KUKA KRL program: MyProgram_127().src

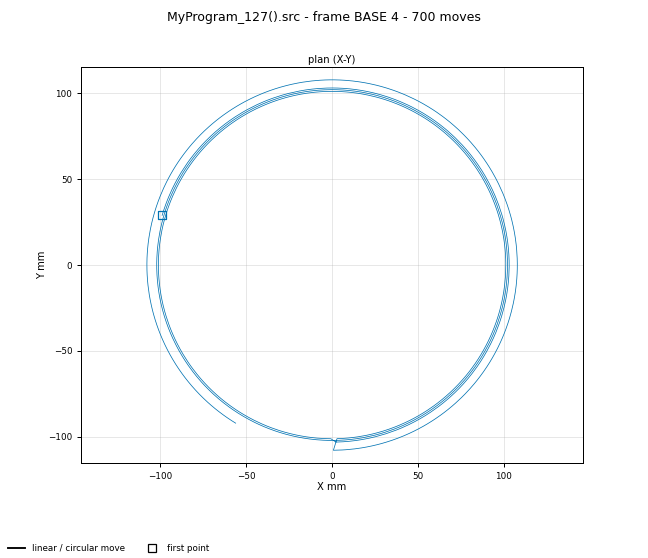
[picture p0: tool path of MyProgram_127().src in frame BASE 4, 700 of 700 moves have a stored position in this frame; points joined in program order, loops and branches not executed]
&ACCESS RVP
&REL 1
&PARAM TEMPLATE = C:\KRC\Roboter\Template\vorgabe
&PARAM EDITMASK = *
DEF MyProgram_127()
; ---- Setting reference (Base) ----
$BASE = BASE_DATA[4]

; --------------------------
; ---- Setting tool (TCP) ----
$TOOL = TOOL_DATA[3]
; --------------------------

$VEL.CP = VEL_APROX_PRINT
Startdeposition()
$VEL.CP = VEL_PRINT
LIN {X -98.9331,Y 28.9212,Z 105,A 158.7425,B 24.9321,C -1.9035,E1 24.8466,E2 286.8295} C_DIS
LIN {X -97.9061,Y 32.2288,Z 105,A 156.9125,B 24.9314,C -1.9128,E1 24.8481,E2 288.6479} C_DIS
LIN {X -96.4517,Y 36.3475,Z 105,A 154.6927,B 24.9303,C -1.9275,E1 24.8502,E2 290.845} C_DIS
LIN {X -95.1957,Y 39.5236,Z 105,A 152.0792,B 24.9317,C -1.9086,E1 24.853,E2 293.5182} C_DIS
LIN {X -93.0833,Y 44.2686,Z 105,A 149.0809,B 24.9314,C -1.9135,E1 24.8565,E2 296.5212} C_DIS
LIN {X -91.5484,Y 47.3623,Z 105,A 147.5482,B 24.93,C -1.9325,E1 24.8584,E2 298.0168} C_DIS
LIN {X -89.8281,Y 50.5476,Z 105,A 145.7731,B 24.929,C -1.9467,E1 24.8608,E2 299.7675} C_DIS
LIN {X -87.9398,Y 53.7652,Z 105,A 143.5022,B 24.929,C -1.9458,E1 24.864,E2 302.0523} C_DIS
LIN {X -84.3049,Y 59.3047,Z 105,A 139.7147,B 24.9285,C -1.9524,E1 24.8699,E2 305.8429} C_DIS
LIN {X -82.5416,Y 61.7331,Z 105,A 138.1139,B 24.928,C -1.9593,E1 24.8726,E2 307.435} C_DIS
LIN {X -80.3974,Y 64.5023,Z 105,A 136.0774,B 24.9279,C -1.9613,E1 24.8761,E2 309.4763} C_DIS
LIN {X -78.1163,Y 67.247,Z 105,A 134.0692,B 24.9276,C -1.9656,E1 24.8797,E2 311.4835} C_DIS
LIN {X -75.6889,Y 69.9669,Z 105,A 132.0269,B 24.9272,C -1.9701,E1 24.8835,E2 313.524} C_DIS
LIN {X -73.2076,Y 72.5583,Z 105,A 130.0602,B 24.9268,C -1.976,E1 24.8874,E2 315.4851} C_DIS
LIN {X -70.5493,Y 75.1455,Z 105,A 128.0084,B 24.9264,C -1.9813,E1 24.8915,E2 317.5329} C_DIS
LIN {X -67.891,Y 77.5556,Z 105,A 126.0734,B 24.9259,C -1.9879,E1 24.8955,E2 319.4598} C_DIS
LIN {X -65.3097,Y 79.7431,Z 105,A 124.0713,B 24.9259,C -1.9879,E1 24.8998,E2 321.4698} C_DIS
LIN {X -62.5207,Y 81.9479,Z 105,A 122.0628,B 24.9257,C -1.9909,E1 24.9043,E2 323.4783} C_DIS
LIN {X -59.7475,Y 83.9899,Z 105,A 120.1946,B 24.9253,C -1.9965,E1 24.9085,E2 325.3398} C_DIS
LIN {X -56.6556,Y 86.1057,Z 105,A 118.0284,B 24.9252,C -1.9976,E1 24.9135,E2 327.5105} C_DIS
LIN {X -52.2933,Y 88.8227,Z 105,A 114.8044,B 24.9258,C -1.9898,E1 24.9213,E2 330.763} C_DIS
LIN {X -49.2603,Y 90.5399,Z 105,A 113.6441,B 24.9234,C -2.0209,E1 24.9239,E2 331.8525} C_DIS
LIN {X -43.6643,Y 93.3676,Z 105,A 109.6852,B 24.9243,C -2.0094,E1 24.9339,E2 335.8492} C_DIS
LIN {X -40.088,Y 94.9579,Z 105,A 107.6299,B 24.9237,C -2.017,E1 24.9392,E2 337.8914} C_DIS
LIN {X -37.8178,Y 95.8847,Z 105,A 105.9153,B 24.9245,C -2.0061,E1 24.9437,E2 339.6355} C_DIS
LIN {X -34.2696,Y 97.2093,Z 105,A 103.2372,B 24.9259,C -1.9882,E1 24.9509,E2 342.3615} C_DIS
LIN {X -29.2299,Y 98.8416,Z 105,A 101.2027,B 24.9232,C -2.0244,E1 24.9561,E2 344.3135} C_DIS
LIN {X -25.3353,Y 99.9113,Z 105,A 97.6855,B 24.9265,C -1.9806,E1 24.9659,E2 347.9399} C_DIS
LIN {X -18.7953,Y 101.3464,Z 105,A 95.1628,B 24.9229,C -2.0271,E1 24.9725,E2 350.3548} C_DIS
LIN {X -15.2046,Y 101.9468,Z 105,A 93.1403,B 24.9229,C -2.0286,E1 24.9781,E2 352.3756} C_DIS
LIN {X -11.8481,Y 102.3898,Z 105,A 91.2817,B 24.9227,C -2.0306,E1 24.9832,E2 354.2308} C_DIS
LIN {X -8.2839,Y 102.7396,Z 105,A 89.3552,B 24.9224,C -2.0339,E1 24.9886,E2 356.1503} C_DIS
LIN {X -2.9459,Y 103.0311,Z 105,A 86.2952,B 24.9226,C -2.0316,E1 24.9971,E2 359.2164} C_DIS
LIN {X 0.2408,Y 103.0734,Z 105,A 84.5977,B 24.9224,C -2.0348,E1 25.0018,E2 360.9065} C_DIS
LIN {X 3.0527,Y 103.0278,Z 105,A 83.223,B 24.9218,C -2.0421,E1 25.0056,E2 362.2637} C_DIS
LIN {X 6.6028,Y 102.8619,Z 105,A 81.0175,B 24.9225,C -2.0334,E1 25.0118,E2 364.4889} C_DIS
LIN {X 10.2822,Y 102.5598,Z 105,A 78.9583,B 24.9225,C -2.033,E1 25.0176,E2 366.5479} C_DIS
LIN {X 13.8719,Y 102.1372,Z 105,A 76.8656,B 24.9228,C -2.0294,E1 25.0234,E2 368.6476} C_DIS
LIN {X 17.6219,Y 101.5574,Z 105,A 74.8,B 24.9228,C -2.0303,E1 25.0291,E2 370.7088} C_DIS
LIN {X 20.3768,Y 101.0394,Z 105,A 73.3018,B 24.9226,C -2.032,E1 25.0331,E2 372.2014} C_DIS
LIN {X 24.0252,Y 100.2347,Z 105,A 70.5318,B 24.9247,C -2.0045,E1 25.0408,E2 375.0326} C_DIS
LIN {X 28.3201,Y 99.1063,Z 105,A 68.8567,B 24.9225,C -2.0331,E1 25.0452,E2 376.6371} C_DIS
LIN {X 32.8253,Y 97.7065,Z 105,A 66.1547,B 24.9229,C -2.0279,E1 25.0524,E2 379.3463} C_DIS
LIN {X 36.3868,Y 96.4368,Z 105,A 64.0979,B 24.9229,C -2.0277,E1 25.0577,E2 381.3992} C_DIS
LIN {X 39.5015,Y 95.205,Z 105,A 62.1207,B 24.9234,C -2.0213,E1 25.0629,E2 383.3872} C_DIS
LIN {X 44.2426,Y 93.0958,Z 105,A 59.3176,B 24.9234,C -2.0212,E1 25.07,E2 386.1837} C_DIS
LIN {X 46.6843,Y 91.8949,Z 105,A 57.7654,B 24.9237,C -2.0177,E1 25.0739,E2 387.7398} C_DIS
LIN {X 49.9449,Y 90.1647,Z 105,A 55.6228,B 24.9241,C -2.0113,E1 25.0792,E2 389.8913} C_DIS
LIN {X 53.2665,Y 88.2429,Z 105,A 53.5728,B 24.9241,C -2.0115,E1 25.0841,E2 391.9348} C_DIS
LIN {X 56.8312,Y 85.9899,Z 105,A 50.8513,B 24.9255,C -1.9929,E1 25.0905,E2 394.6912} C_DIS
LIN {X 59.7089,Y 84.0174,Z 105,A 49.4236,B 24.9243,C -2.0098,E1 25.0937,E2 396.074} C_DIS
LIN {X 62.6655,Y 81.8362,Z 105,A 47.3819,B 24.9245,C -2.0062,E1 25.0983,E2 398.1169} C_DIS
LIN {X 65.6264,Y 79.4816,Z 105,A 45.2669,B 24.9249,C -2.0018,E1 25.1029,E2 400.2343} C_DIS
LIN {X 67.4456,Y 77.9445,Z 105,A 42.9443,B 24.928,C -1.9596,E1 25.108,E2 402.6473} C_DIS
LIN {X 71.5189,Y 74.2233,Z 105,A 40.883,B 24.9255,C -1.9931,E1 25.1119,E2 404.621} C_DIS
LIN {X 75.7947,Y 69.8516,Z 105,A 37.5,B 24.926,C -1.9863,E1 25.1185,E2 408.0055} C_DIS
LIN {X 78.1453,Y 67.2129,Z 105,A 35.7185,B 24.9258,C -1.9892,E1 25.1217,E2 409.7722} C_DIS
LIN {X 80.4406,Y 64.4491,Z 105,A 33.6595,B 24.9263,C -1.982,E1 25.1254,E2 411.8389} C_DIS
LIN {X 82.9467,Y 61.1884,Z 105,A 31.2667,B 24.9271,C -1.972,E1 25.1295,E2 414.2437} C_DIS
LIN {X 84.7752,Y 58.6283,Z 105,A 29.304,B 24.9281,C -1.959,E1 25.1326,E2 416.2276} C_DIS
LIN {X 87.1111,Y 55.1002,Z 105,A 27.1308,B 24.928,C -1.9601,E1 25.1359,E2 418.3873} C_DIS
LIN {X 89.1835,Y 51.6762,Z 105,A 24.7081,B 24.929,C -1.9461,E1 25.1394,E2 420.8305} C_DIS
LIN {X 91.4934,Y 47.47,Z 105,A 22.2461,B 24.929,C -1.9471,E1 25.1426,E2 423.2772} C_DIS
LIN {X 93.2653,Y 43.884,Z 105,A 19.9203,B 24.9297,C -1.9367,E1 25.1454,E2 425.6151} C_DIS
LIN {X 95.0509,Y 39.8672,Z 105,A 17.6491,B 24.9297,C -1.9367,E1 25.1479,E2 427.8739} C_DIS
LIN {X 97.0088,Y 34.8366,Z 105,A 14.491,B 24.9308,C -1.9214,E1 25.1511,E2 431.0506} C_DIS
LIN {X 98.7758,Y 29.4516,Z 105,A 11.6761,B 24.9305,C -1.9257,E1 25.1534,E2 433.8393} C_DIS
LIN {X 99.4228,Y 27.1889,Z 105,A 10.1237,B 24.9315,C -1.9116,E1 25.1546,E2 435.416} C_DIS
LIN {X 100.4196,Y 23.2365,Z 105,A 8.0347,B 24.9315,C -1.9119,E1 25.156,E2 437.4922} C_DIS
LIN {X 101.1933,Y 19.5951,Z 105,A 6.011,B 24.9318,C -1.9073,E1 25.1571,E2 439.5149} C_DIS
LIN {X 101.766,Y 16.3743,Z 105,A 4.0964,B 24.9325,C -1.8976,E1 25.158,E2 441.4412} C_DIS
LIN {X 102.2145,Y 13.2757,Z 105,A 2.4368,B 24.9326,C -1.8955,E1 25.1586,E2 443.0961} C_DIS
LIN {X 102.6055,Y 9.8116,Z 105,A 0.2998,B 24.9337,C -1.881,E1 25.1592,E2 445.2545} C_DIS
LIN {X 102.8922,Y 6.1161,Z 105,A -2.0033,B 24.9348,C -1.8644,E1 25.1597,E2 447.5831} C_DIS
LIN {X 103.0443,Y 2.5058,Z 105,A -3.5818,B 24.9341,C -1.8756,E1 25.1597,E2 449.1257} C_DIS
LIN {X 103.0694,Y -0.9185,Z 105,A -5.6826,B 24.9351,C -1.8613,E1 25.1597,E2 451.2477} C_DIS
LIN {X 102.8757,Y -6.3964,Z 105,A -8.5358,B 24.9351,C -1.8595,E1 25.1594,E2 454.0884} C_DIS
LIN {X 102.5639,Y -10.2437,Z 105,A -10.6155,B 24.9355,C -1.8553,E1 25.1589,E2 456.1656} C_DIS
LIN {X 102.2015,Y -13.3755,Z 105,A -12.9205,B 24.9374,C -1.8268,E1 25.158,E2 458.5242} C_DIS
LIN {X 101.5816,Y -17.4772,Z 105,A -14.6875,B 24.9364,C -1.8416,E1 25.1572,E2 460.246} C_DIS
LIN {X 101.006,Y -20.5391,Z 105,A -16.9672,B 24.9384,C -1.8134,E1 25.1559,E2 462.5787} C_DIS
LIN {X 100.0741,Y -24.6836,Z 105,A -18.9962,B 24.9379,C -1.8196,E1 25.1546,E2 464.5816} C_DIS
LIN {X 98.6723,Y -29.8005,Z 105,A -22.1502,B 24.9392,C -1.8018,E1 25.1521,E2 467.7594} C_DIS
LIN {X 97.4856,Y -33.4781,Z 105,A -23.7692,B 24.9381,C -1.8169,E1 25.1507,E2 469.3337} C_DIS
LIN {X 95.3975,Y -39.0306,Z 105,A -27.0314,B 24.9387,C -1.8081,E1 25.1474,E2 472.5984} C_DIS
LIN {X 94.0262,Y -42.2271,Z 105,A -28.9192,B 24.939,C -1.8041,E1 25.1453,E2 474.4854} C_DIS
LIN {X 92.3169,Y -45.8435,Z 105,A -31.9753,B 24.9417,C -1.7633,E1 25.1415,E2 477.6214} C_DIS
LIN {X 89.9827,Y -50.2708,Z 105,A -33.8915,B 24.9399,C -1.7906,E1 25.139,E2 479.4632} C_DIS
LIN {X 88.182,Y -53.3668,Z 105,A -35.8602,B 24.9402,C -1.7857,E1 25.1362,E2 481.4332} C_DIS
LIN {X 86.3032,Y -56.3561,Z 105,A -37.8502,B 24.9407,C -1.779,E1 25.1332,E2 483.4292} C_DIS
LIN {X 84.321,Y -59.2816,Z 105,A -39.6571,B 24.9407,C -1.78,E1 25.1303,E2 485.2248} C_DIS
LIN {X 81.5215,Y -63.0739,Z 105,A -42.4647,B 24.9416,C -1.7652,E1 25.1256,E2 488.054} C_DIS
LIN {X 79.3093,Y -65.8337,Z 105,A -44.315,B 24.9416,C -1.7647,E1 25.1223,E2 489.8968} C_DIS
LIN {X 76.2926,Y -69.309,Z 105,A -47.3279,B 24.9433,C -1.7396,E1 25.1167,E2 492.9556} C_DIS
LIN {X 73.9687,Y -71.783,Z 105,A -48.8527,B 24.9426,C -1.7496,E1 25.1138,E2 494.4501} C_DIS
LIN {X 71.4083,Y -74.3298,Z 105,A -50.6769,B 24.9425,C -1.7522,E1 25.1102,E2 496.2605} C_DIS
LIN {X 68.2586,Y -77.2345,Z 105,A -53.4557,B 24.9439,C -1.7305,E1 25.1043,E2 499.0795} C_DIS
LIN {X 64.8251,Y -80.1359,Z 105,A -55.5771,B 24.9432,C -1.7402,E1 25.0998,E2 501.1697} C_DIS
LIN {X 61.9703,Y -82.3634,Z 105,A -57.4686,B 24.9432,C -1.7408,E1 25.0957,E2 503.0529} C_DIS
LIN {X 57.4935,Y -85.5491,Z 105,A -60.7281,B 24.9442,C -1.7263,E1 25.0882,E2 506.3356} C_DIS
LIN {X 54.3113,Y -87.6039,Z 105,A -62.8267,B 24.9444,C -1.7225,E1 25.0832,E2 508.4363} C_DIS
LIN {X 51.2517,Y -89.4277,Z 105,A -64.7594,B 24.9445,C -1.7208,E1 25.0785,E2 510.3671} C_DIS
LIN {X 48.1624,Y -91.1287,Z 105,A -66.8295,B 24.945,C -1.713,E1 25.0734,E2 512.4498} C_DIS
LIN {X 44.5578,Y -92.9443,Z 105,A -69.156,B 24.9455,C -1.706,E1 25.0676,E2 514.7866} C_DIS
LIN {X 40.2998,Y -94.8686,Z 105,A -71.5025,B 24.9451,C -1.7121,E1 25.0616,E2 517.113} C_DIS
LIN {X 37.386,Y -96.0543,Z 105,A -73.0986,B 24.9448,C -1.7157,E1 25.0575,E2 518.697} C_DIS
LIN {X 31.3492,Y -98.1908,Z 105,A -76.7392,B 24.9453,C -1.7079,E1 25.0479,E2 522.3488} C_DIS
LIN {X 25.1272,Y -99.9648,Z 105,A -80.4693,B 24.9459,C -1.6987,E1 25.0378,E2 526.0946} C_DIS
LIN {X 21.5396,Y -100.7982,Z 105,A -82.6382,B 24.9463,C -1.692,E1 25.0318,E2 528.2763} C_DIS
LIN {X 17.2353,Y -101.622,Z 105,A -84.8606,B 24.9459,C -1.6984,E1 25.0258,E2 530.4811} C_DIS
LIN {X 13.9298,Y -102.129,Z 105,A -86.6561,B 24.9459,C -1.6996,E1 25.0208,E2 532.2723} C_DIS
LIN {X 10.2271,Y -102.5656,Z 105,A -88.8876,B 24.9463,C -1.6922,E1 25.0146,E2 534.5198} C_DIS
LIN {X 6.5489,Y -102.8655,Z 105,A -90.789,B 24.946,C -1.6971,E1 25.0093,E2 536.4087} C_DIS
LIN {X 2.2675,Y -103.0487,Z 105,A -93.5057,B 24.9469,C -1.6834,E1 25.0017,E2 539.1572} C_DIS
LIN {X 2.2675,Y -103.0487,Z 105,A -93.5057,B 24.9469,C -1.6834,E1 25.0017,E2 539.1572} C_DIS
Enddeposition()
LIN {X 0.721,Y -102.0888,Z 105,A -93.9703,B 24.9448,C -1.7156,E1 25.0006,E2 539.5454} C_DIS
Startdeposition()
$VEL.CP = VEL_PRINT
LIN {X 4.1196,Y -102.0095,Z 105,A -91.4318,B 24.9432,C -1.7405,E1 25.0078,E2 536.9484} C_DIS
LIN {X 7.4303,Y -101.8231,Z 105,A -89.3693,B 24.9427,C -1.7491,E1 25.0136,E2 534.8663} C_DIS
LIN {X 11.0426,Y -101.4942,Z 105,A -87.3963,B 24.9427,C -1.7478,E1 25.0191,E2 532.8977} C_DIS
LIN {X 14.4327,Y -101.0671,Z 105,A -85.549,B 24.9428,C -1.7463,E1 25.0242,E2 531.0555} C_DIS
LIN {X 18.1999,Y -100.4571,Z 105,A -83.3169,B 24.9425,C -1.7515,E1 25.0304,E2 528.8133} C_DIS
LIN {X 24.5658,Y -99.0935,Z 105,A -79.2947,B 24.9413,C -1.7696,E1 25.0414,E2 524.7539} C_DIS
LIN {X 27.8744,Y -98.2134,Z 105,A -77.4471,B 24.9413,C -1.7687,E1 25.0464,E2 522.9113} C_DIS
LIN {X 30.9944,Y -97.2749,Z 105,A -76.2081,B 24.9428,C -1.7474,E1 25.0495,E2 521.7251} C_DIS
LIN {X 35.848,Y -95.5922,Z 105,A -73.3976,B 24.9428,C -1.7483,E1 25.0569,E2 518.9183} C_DIS
LIN {X 38.3912,Y -94.599,Z 105,A -71.6044,B 24.9419,C -1.7608,E1 25.0616,E2 517.0994} C_DIS
LIN {X 41.6475,Y -93.2118,Z 105,A -69.6571,B 24.9418,C -1.7622,E1 25.0666,E2 515.1534} C_DIS
LIN {X 45.3721,Y -91.4561,Z 105,A -67.3176,B 24.9415,C -1.7671,E1 25.0725,E2 512.8086} C_DIS
LIN {X 48.6468,Y -89.7571,Z 105,A -65.2945,B 24.9414,C -1.7688,E1 25.0775,E2 510.7873} C_DIS
LIN {X 51.7894,Y -87.9815,Z 105,A -63.1915,B 24.9409,C -1.7755,E1 25.0826,E2 508.6746} C_DIS
LIN {X 55.0242,Y -85.9954,Z 105,A -61.1724,B 24.9409,C -1.7751,E1 25.0874,E2 506.6629} C_DIS
LIN {X 57.6899,Y -84.232,Z 105,A -59.1419,B 24.9401,C -1.7883,E1 25.0921,E2 504.6081} C_DIS
LIN {X 61.1906,Y -81.7226,Z 105,A -56.9001,B 24.9401,C -1.7862,E1 25.0972,E2 502.3792} C_DIS
LIN {X 64.102,Y -79.4596,Z 105,A -54.8901,B 24.9401,C -1.7883,E1 25.1015,E2 500.3717} C_DIS
LIN {X 66.6309,Y -77.353,Z 105,A -52.9286,B 24.9395,C -1.7972,E1 25.1058,E2 498.3969} C_DIS
LIN {X 69.4854,Y -74.7996,Z 105,A -50.8033,B 24.9392,C -1.8012,E1 25.1101,E2 496.2707} C_DIS
LIN {X 72.0356,Y -72.3456,Z 105,A -48.8262,B 24.9389,C -1.8057,E1 25.1141,E2 494.2913} C_DIS
LIN {X 74.6311,Y -69.6649,Z 105,A -46.7222,B 24.9385,C -1.8113,E1 25.1181,E2 492.1831} C_DIS
LIN {X 77.1023,Y -66.9192,Z 105,A -44.7019,B 24.9383,C -1.8145,E1 25.1219,E2 490.1644} C_DIS
LIN {X 79.3841,Y -64.1952,Z 105,A -42.7562,B 24.9381,C -1.8178,E1 25.1253,E2 488.2199} C_DIS
LIN {X 81.7271,Y -61.1846,Z 105,A -40.6159,B 24.9377,C -1.8235,E1 25.1289,E2 486.0763} C_DIS
LIN {X 83.2512,Y -59.0943,Z 105,A -39.1653,B 24.9374,C -1.8275,E1 25.1313,E2 484.6234} C_DIS
LIN {X 85.2746,Y -56.1346,Z 105,A -37.2939,B 24.9374,C -1.8273,E1 25.1342,E2 482.7616} C_DIS
LIN {X 87.1032,Y -53.2536,Z 105,A -35.3038,B 24.9368,C -1.8359,E1 25.1371,E2 480.7614} C_DIS
LIN {X 88.8211,Y -50.3391,Z 105,A -33.0561,B 24.9354,C -1.8559,E1 25.1403,E2 478.478} C_DIS
LIN {X 91.0686,Y -46.1463,Z 105,A -30.9367,B 24.9365,C -1.841,E1 25.143,E2 476.4051} C_DIS
LIN {X 92.2699,Y -43.6973,Z 105,A -29.3302,B 24.9359,C -1.8487,E1 25.145,E2 474.789} C_DIS
LIN {X 93.6815,Y -40.5793,Z 105,A -27.4588,B 24.9357,C -1.8525,E1 25.1471,E2 472.9188} C_DIS
LIN {X 94.8687,Y -37.7222,Z 105,A -25.5424,B 24.9348,C -1.8653,E1 25.1491,E2 470.9827} C_DIS
LIN {X 96.0625,Y -34.5694,Z 105,A -23.6623,B 24.9344,C -1.8707,E1 25.1509,E2 469.1004} C_DIS
LIN {X 97.9024,Y -28.9477,Z 105,A -20.9212,B 24.9354,C -1.8571,E1 25.1533,E2 466.407} C_DIS
LIN {X 99.1832,Y -24.1978,Z 105,A -17.079,B 24.9315,C -1.911,E1 25.156,E2 462.4599} C_DIS
LIN {X 100.0882,Y -20.1338,Z 105,A -15.3316,B 24.9328,C -1.8937,E1 25.157,E2 460.7633} C_DIS
LIN {X 100.7051,Y -16.7728,Z 105,A -13.3231,B 24.9321,C -1.9037,E1 25.1579,E2 458.7431} C_DIS
LIN {X 101.2353,Y -13.2015,Z 105,A -11.5637,B 24.9324,C -1.8991,E1 25.1586,E2 457.0049} C_DIS
LIN {X 101.5747,Y -10.2741,Z 105,A -9.9269,B 24.9321,C -1.9038,E1 25.1591,E2 455.3668} C_DIS
LIN {X 101.8511,Y -7.0152,Z 105,A -7.9723,B 24.9313,C -1.9147,E1 25.1595,E2 453.398} C_DIS
LIN {X 102.0386,Y -3.3166,Z 105,A -5.934,B 24.9309,C -1.9197,E1 25.1597,E2 451.3599} C_DIS
LIN {X 102.0935,Y 0.1526,Z 105,A -3.9243,B 24.9303,C -1.9286,E1 25.1597,E2 449.3413} C_DIS
LIN {X 102.0323,Y 3.5243,Z 105,A -1.9696,B 24.9296,C -1.9373,E1 25.1597,E2 447.3776} C_DIS
LIN {X 101.8489,Y 7.0485,Z 105,A -0.1682,B 24.9297,C -1.9362,E1 25.1593,E2 445.5895} C_DIS
LIN {X 101.5483,Y 10.5265,Z 105,A 1.7807,B 24.9293,C -1.942,E1 25.1588,E2 443.6384} C_DIS
LIN {X 101.1877,Y 13.5688,Z 105,A 3.5191,B 24.9288,C -1.9483,E1 25.1582,E2 441.8956} C_DIS
LIN {X 100.6848,Y 16.8944,Z 105,A 5.3429,B 24.9286,C -1.9516,E1 25.1574,E2 440.0746} C_DIS
LIN {X 100.0225,Y 20.4539,Z 105,A 7.3093,B 24.9283,C -1.9553,E1 25.1563,E2 438.1111} C_DIS
LIN {X 99.3482,Y 23.5179,Z 105,A 9.2116,B 24.9275,C -1.9666,E1 25.1551,E2 436.1932} C_DIS
LIN {X 98.0107,Y 28.5826,Z 105,A 11.8721,B 24.9277,C -1.964,E1 25.1532,E2 433.5541} C_DIS
LIN {X 95.6853,Y 35.6022,Z 105,A 16.2496,B 24.9261,C -1.9857,E1 25.1493,E2 429.15} C_DIS
LIN {X 94.3586,Y 38.9819,Z 105,A 18.2975,B 24.9256,C -1.9921,E1 25.1471,E2 427.0984} C_DIS
LIN {X 92.869,Y 42.4079,Z 105,A 20.3571,B 24.9253,C -1.9965,E1 25.1448,E2 425.0395} C_DIS
LIN {X 91.3792,Y 45.5273,Z 105,A 22.2975,B 24.9248,C -2.002,E1 25.1424,E2 423.0965} C_DIS
LIN {X 89.5981,Y 48.94,Z 105,A 24.2486,B 24.925,C -1.9994,E1 25.1398,E2 421.1619} C_DIS
LIN {X 87.3824,Y 52.7944,Z 105,A 26.5561,B 24.9251,C -1.9984,E1 25.1366,E2 418.8686} C_DIS
LIN {X 86.0424,Y 54.951,Z 105,A 28.3625,B 24.9237,C -2.0177,E1 25.1339,E2 417.0257} C_DIS
LIN {X 83.7233,Y 58.4233,Z 105,A 30.4233,B 24.9241,C -2.0122,E1 25.1307,E2 414.9882} C_DIS
LIN {X 82.2523,Y 60.4769,Z 105,A 32.0058,B 24.9233,C -2.0224,E1 25.128,E2 413.3892} C_DIS
LIN {X 80.1709,Y 63.2099,Z 105,A 33.9308,B 24.923,C -2.027,E1 25.1247,E2 411.4625} C_DIS
LIN {X 77.7176,Y 66.2029,Z 105,A 35.889,B 24.9232,C -2.0234,E1 25.1213,E2 409.5216} C_DIS
LIN {X 75.9732,Y 68.1978,Z 105,A 37.523,B 24.9225,C -2.0327,E1 25.1182,E2 407.873} C_DIS
LIN {X 73.0332,Y 71.3395,Z 105,A 39.8316,B 24.9225,C -2.0337,E1 25.1138,E2 405.572} C_DIS
LIN {X 70.1295,Y 74.1942,Z 105,A 42.2617,B 24.9216,C -2.0444,E1 25.1089,E2 403.1269} C_DIS
LIN {X 66.5865,Y 77.3908,Z 105,A 44.735,B 24.9218,C -2.0415,E1 25.1038,E2 400.6703} C_DIS
LIN {X 63.6644,Y 79.8117,Z 105,A 46.9834,B 24.9212,C -2.0503,E1 25.0989,E2 398.4097} C_DIS
LIN {X 61.2434,Y 81.6829,Z 105,A 48.6719,B 24.921,C -2.0522,E1 25.0951,E2 396.7227} C_DIS
LIN {X 58.9121,Y 83.3812,Z 105,A 50.57,B 24.9199,C -2.0661,E1 25.0908,E2 394.7984} C_DIS
LIN {X 55.159,Y 85.9089,Z 105,A 52.9287,B 24.9202,C -2.063,E1 25.0853,E2 392.4549} C_DIS
LIN {X 52.0441,Y 87.831,Z 105,A 54.9631,B 24.92,C -2.0653,E1 25.0804,E2 390.4214} C_DIS
LIN {X 48.2339,Y 89.9811,Z 105,A 57.6131,B 24.9192,C -2.0764,E1 25.0739,E2 387.7528} C_DIS
LIN {X 45.1767,Y 91.553,Z 105,A 59.3615,B 24.9195,C -2.0717,E1 25.0696,E2 386.0202} C_DIS
LIN {X 41.7531,Y 93.1642,Z 105,A 61.2605,B 24.92,C -2.0654,E1 25.0648,E2 384.1409} C_DIS
LIN {X 39.2802,Y 94.2341,Z 105,A 62.8299,B 24.9197,C -2.0692,E1 25.0608,E2 382.5661} C_DIS
LIN {X 36.4723,Y 95.3558,Z 105,A 64.6333,B 24.9193,C -2.0751,E1 25.0561,E2 380.7529} C_DIS
LIN {X 33.3696,Y 96.4859,Z 105,A 66.5192,B 24.919,C -2.078,E1 25.0511,E2 378.864} C_DIS
LIN {X 29.9778,Y 97.5923,Z 105,A 68.4737,B 24.919,C -2.0777,E1 25.0459,E2 376.9136} C_DIS
LIN {X 26.5895,Y 98.569,Z 105,A 70.3895,B 24.9191,C -2.0766,E1 25.0408,E2 375.0037} C_DIS
LIN {X 23.5975,Y 99.3297,Z 105,A 72.0695,B 24.9192,C -2.0756,E1 25.0362,E2 373.3286} C_DIS
LIN {X 19.4478,Y 100.223,Z 105,A 74.205,B 24.9199,C -2.0673,E1 25.0305,E2 371.2155} C_DIS
LIN {X 16.9671,Y 100.6727,Z 105,A 75.9633,B 24.9188,C -2.0809,E1 25.0255,E2 369.4268} C_DIS
LIN {X 13.4123,Y 101.2079,Z 105,A 78.013,B 24.9187,C -2.0827,E1 25.0198,E2 367.3747} C_DIS
LIN {X 9.9806,Y 101.6051,Z 105,A 79.9511,B 24.9187,C -2.0829,E1 25.0145,E2 365.4374} C_DIS
LIN {X 6.5414,Y 101.8832,Z 105,A 81.9106,B 24.9186,C -2.0839,E1 25.009,E2 363.4765} C_DIS
LIN {X 2.7045,Y 102.0574,Z 105,A 83.9174,B 24.919,C -2.0781,E1 25.0034,E2 361.484} C_DIS
LIN {X -0.6181,Y 102.0905,Z 105,A 85.9275,B 24.9186,C -2.0832,E1 24.9978,E2 359.4617} C_DIS
LIN {X -4.5435,Y 101.9913,Z 105,A 88.1515,B 24.9186,C -2.0832,E1 24.9916,E2 357.2372} C_DIS
LIN {X -8.2012,Y 101.7624,Z 105,A 90.1031,B 24.919,C -2.0785,E1 24.9862,E2 355.2963} C_DIS
LIN {X -11.507,Y 101.4425,Z 105,A 92.038,B 24.9189,C -2.0801,E1 24.9808,E2 353.3563} C_DIS
LIN {X -15.0669,Y 100.9759,Z 105,A 94.1185,B 24.9188,C -2.0813,E1 24.975,E2 351.2714} C_DIS
LIN {X -18.6514,Y 100.3759,Z 105,A 96.6062,B 24.9176,C -2.0964,E1 24.9681,E2 348.7453} C_DIS
LIN {X -22.2866,Y 99.6316,Z 105,A 98.0528,B 24.9196,C -2.071,E1 24.9643,E2 347.3573} C_DIS
LIN {X -25.4244,Y 98.8759,Z 105,A 99.9697,B 24.9194,C -2.0731,E1 24.9591,E2 345.4325} C_DIS
LIN {X -28.7193,Y 97.9702,Z 105,A 101.8852,B 24.9196,C -2.071,E1 24.954,E2 343.519} C_DIS
LIN {X -31.5861,Y 97.0835,Z 105,A 103.8842,B 24.9188,C -2.0806,E1 24.9486,E2 341.4937} C_DIS
LIN {X -35.2296,Y 95.8217,Z 105,A 105.8472,B 24.9196,C -2.0704,E1 24.9435,E2 339.5509} C_DIS
LIN {X -38.7091,Y 94.4696,Z 105,A 107.7678,B 24.9203,C -2.0612,E1 24.9385,E2 337.6481} C_DIS
LIN {X -41.5395,Y 93.2605,Z 105,A 109.6254,B 24.9202,C -2.0634,E1 24.9337,E2 335.7808} C_DIS
LIN {X -45.6434,Y 91.3216,Z 105,A 112.1218,B 24.9206,C -2.0575,E1 24.9275,E2 333.292} C_DIS
LIN {X -48.8645,Y 89.639,Z 105,A 114.2546,B 24.9206,C -2.0575,E1 24.9222,E2 331.1533} C_DIS
LIN {X -51.8921,Y 87.9208,Z 105,A 116.1167,B 24.9211,C -2.0507,E1 24.9177,E2 329.3019} C_DIS
LIN {X -56.924,Y 84.7505,Z 105,A 119.5287,B 24.9214,C -2.0469,E1 24.9097,E2 325.8878} C_DIS
LIN {X -59.619,Y 82.8769,Z 105,A 121.3731,B 24.9217,C -2.0433,E1 24.9055,E2 324.0457} C_DIS
LIN {X -62.2181,Y 80.943,Z 105,A 123.1864,B 24.922,C -2.0393,E1 24.9015,E2 322.2354} C_DIS
LIN {X -64.9402,Y 78.7767,Z 105,A 125.1815,B 24.9222,C -2.0365,E1 24.8972,E2 320.2394} C_DIS
LIN {X -67.6757,Y 76.4406,Z 105,A 127.2649,B 24.9224,C -2.0342,E1 24.8928,E2 318.1532} C_DIS
LIN {X -70.3797,Y 73.9588,Z 105,A 129.3562,B 24.9227,C -2.0305,E1 24.8885,E2 316.0623} C_DIS
LIN {X -73.0796,Y 71.2924,Z 105,A 131.493,B 24.9231,C -2.0256,E1 24.8843,E2 313.9281} C_DIS
LIN {X -75.5845,Y 68.6302,Z 105,A 133.5407,B 24.9235,C -2.0203,E1 24.8804,E2 311.8839} C_DIS
LIN {X -78.0791,Y 65.7786,Z 105,A 135.6516,B 24.9239,C -2.0143,E1 24.8766,E2 309.7777} C_DIS
LIN {X -80.3533,Y 62.9791,Z 105,A 137.6353,B 24.9244,C -2.0075,E1 24.8732,E2 307.8009} C_DIS
LIN {X -82.4193,Y 60.2488,Z 105,A 139.4785,B 24.925,C -1.9996,E1 24.8701,E2 305.9677} C_DIS
LIN {X -84.9711,Y 56.5936,Z 105,A 142.5184,B 24.9241,C -2.0115,E1 24.8653,E2 302.8843} C_DIS
LIN {X -86.8147,Y 53.7237,Z 105,A 144.215,B 24.9251,C -1.9984,E1 24.8628,E2 301.2102} C_DIS
LIN {X -88.94,Y 50.1267,Z 105,A 146.3959,B 24.9261,C -1.9859,E1 24.8598,E2 299.0479} C_DIS
LIN {X -90.5542,Y 47.1489,Z 105,A 148.7162,B 24.9254,C -1.995,E1 24.8567,E2 296.6936} C_DIS
LIN {X -92.0301,Y 44.1962,Z 105,A 151.1461,B 24.9243,C -2.0098,E1 24.8538,E2 294.2151} C_DIS
LIN {X -94.3244,Y 39.0657,Z 105,A 153.2041,B 24.9278,C -1.9617,E1 24.8517,E2 292.2604} C_DIS
LIN {X -95.3957,Y 36.367,Z 105,A 154.9687,B 24.9278,C -1.9614,E1 24.8498,E2 290.4867} C_DIS
LIN {X -96.2987,Y 33.9032,Z 105,A 156.4532,B 24.9282,C -1.9572,E1 24.8485,E2 289.0038} C_DIS
LIN {X -97.3836,Y 30.6507,Z 105,A 158.4433,B 24.9285,C -1.9535,E1 24.8467,E2 287.0112} C_DIS
LIN {X -98.4559,Y 27.0083,Z 105,A 160.5141,B 24.9291,C -1.9447,E1 24.8452,E2 284.9494} C_DIS
LIN {X -99.2292,Y 24.0095,Z 105,A 162.3087,B 24.9294,C -1.9411,E1 24.844,E2 283.1528} C_DIS
LIN {X -100.1924,Y 19.6069,Z 105,A 164.6019,B 24.9305,C -1.9249,E1 24.8427,E2 280.8848} C_DIS
LIN {X -101.0306,Y 14.6892,Z 105,A 168.3192,B 24.9289,C -1.9478,E1 24.841,E2 277.0907} C_DIS
LIN {X -101.5566,Y 10.4472,Z 105,A 169.8653,B 24.9316,C -1.9103,E1 24.8406,E2 275.6248} C_DIS
LIN {X -101.7838,Y 7.934,Z 105,A 171.5492,B 24.9312,C -1.915,E1 24.8402,E2 273.9196} C_DIS
LIN {X -102.0058,Y 4.2079,Z 105,A 173.556,B 24.932,C -1.9052,E1 24.8399,E2 271.9241} C_DIS
LIN {X -102.088,Y 1.0321,Z 105,A 175.411,B 24.9322,C -1.9019,E1 24.8398,E2 270.0657} C_DIS
LIN {X -102.0704,Y -2.1296,Z 105,A 177.2719,B 24.9324,C -1.8992,E1 24.8398,E2 268.2} C_DIS
LIN {X -101.9303,Y -5.7519,Z 105,A 179.2422,B 24.933,C -1.8905,E1 24.8401,E2 266.2388} C_DIS
LIN {X -101.6541,Y -9.4493,Z 105,A -178.7278,B 24.9336,C -1.882,E1 24.8406,E2 264.2166} C_DIS
LIN {X -101.2936,Y -12.7509,Z 105,A -176.7764,B 24.9338,C -1.8791,E1 24.8412,E2 262.2605} C_DIS
LIN {X -100.828,Y -16.0231,Z 105,A -174.5128,B 24.9332,C -1.8876,E1 24.8422,E2 259.9633} C_DIS
LIN {X -100.2658,Y -19.2254,Z 105,A -173.119,B 24.9347,C -1.8668,E1 24.8429,E2 258.6109} C_DIS
LIN {X -99.5485,Y -22.6508,Z 105,A -170.793,B 24.9342,C -1.8734,E1 24.8443,E2 256.2555} C_DIS
LIN {X -98.5577,Y -26.6313,Z 105,A -168.8538,B 24.9356,C -1.8536,E1 24.8457,E2 254.3521} C_DIS
LIN {X -97.6338,Y -29.8438,Z 105,A -166.8661,B 24.9357,C -1.8518,E1 24.8473,E2 252.3573} C_DIS
LIN {X -96.3946,Y -33.6299,Z 105,A -164.7733,B 24.9365,C -1.8401,E1 24.8491,E2 250.2803} C_DIS
LIN {X -95.2532,Y -36.7432,Z 105,A -162.7204,B 24.9365,C -1.8414,E1 24.8511,E2 248.2129} C_DIS
LIN {X -94.0955,Y -39.6093,Z 105,A -161.0878,B 24.937,C -1.8328,E1 24.8529,E2 246.5917} C_DIS
LIN {X -92.7277,Y -42.7152,Z 105,A -158.9204,B 24.9368,C -1.8366,E1 24.8554,E2 244.4034} C_DIS
LIN {X -90.8084,Y -46.6555,Z 105,A -156.6367,B 24.9377,C -1.8235,E1 24.8582,E2 242.1385} C_DIS
LIN {X -89.065,Y -49.9029,Z 105,A -154.5605,B 24.938,C -1.8182,E1 24.861,E2 240.0641} C_DIS
LIN {X -87.2585,Y -52.9982,Z 105,A -152.6027,B 24.9385,C -1.8109,E1 24.8638,E2 238.1135} C_DIS
LIN {X -85.4427,Y -55.8797,Z 105,A -150.6467,B 24.9388,C -1.8075,E1 24.8667,E2 236.1557} C_DIS
LIN {X -83.6595,Y -58.515,Z 105,A -148.1008,B 24.9372,C -1.8303,E1 24.8709,E2 233.543} C_DIS
LIN {X -81.003,Y -62.1402,Z 105,A -146.6143,B 24.9401,C -1.787,E1 24.8733,E2 232.1527} C_DIS
LIN {X -78.9378,Y -64.7458,Z 105,A -144.3091,B 24.9394,C -1.7982,E1 24.8774,E2 229.8099} C_DIS
LIN {X -76.2513,Y -67.8872,Z 105,A -142.1123,B 24.94,C -1.7885,E1 24.8814,E2 227.6263} C_DIS
LIN {X -74.1803,Y -70.1442,Z 105,A -140.3229,B 24.9401,C -1.7872,E1 24.8848,E2 225.8321} C_DIS
LIN {X -71.6966,Y -72.6805,Z 105,A -138.4202,B 24.9406,C -1.7798,E1 24.8885,E2 223.9391} C_DIS
LIN {X -69.0099,Y -75.2362,Z 105,A -136.2754,B 24.9408,C -1.7778,E1 24.8929,E2 221.7902} C_DIS
LIN {X -66.1528,Y -77.7603,Z 105,A -134.1493,B 24.9411,C -1.7732,E1 24.8974,E2 219.6667} C_DIS
LIN {X -63.3522,Y -80.0585,Z 105,A -132.0701,B 24.9412,C -1.7711,E1 24.9019,E2 217.5847} C_DIS
LIN {X -59.8795,Y -82.6896,Z 105,A -129.5848,B 24.9414,C -1.7683,E1 24.9075,E2 215.0973} C_DIS
LIN {X -57.3802,Y -84.4416,Z 105,A -127.9011,B 24.9417,C -1.7644,E1 24.9113,E2 213.4171} C_DIS
LIN {X -54.8059,Y -86.1355,Z 105,A -126.2697,B 24.9421,C -1.7581,E1 24.9151,E2 211.7955} C_DIS
LIN {X -51.6975,Y -88.0358,Z 105,A -124.1871,B 24.9421,C -1.7565,E1 24.9201,E2 209.7103} C_DIS
LIN {X -48.4186,Y -89.8809,Z 105,A -121.9235,B 24.942,C -1.7592,E1 24.9257,E2 207.4336} C_DIS
LIN {X -45.058,Y -91.6118,Z 105,A -120.0202,B 24.9427,C -1.7485,E1 24.9304,E2 205.5508} C_DIS
LIN {X -42.6038,Y -92.7796,Z 105,A -118.449,B 24.9427,C -1.7484,E1 24.9344,E2 203.9758} C_DIS
LIN {X -39.8062,Y -94.0125,Z 105,A -116.7055,B 24.9427,C -1.7476,E1 24.9388,E2 202.2301} C_DIS
LIN {X -36.9972,Y -95.1534,Z 105,A -114.954,B 24.9427,C -1.7478,E1 24.9434,E2 200.4744} C_DIS
LIN {X -33.1989,Y -96.5456,Z 105,A -112.5788,B 24.9427,C -1.7497,E1 24.9497,E2 198.0898} C_DIS
LIN {X -30.1876,Y -97.5272,Z 105,A -110.9087,B 24.943,C -1.7444,E1 24.9541,E2 196.4294} C_DIS
LIN {X -26.7511,Y -98.5253,Z 105,A -109.0512,B 24.9434,C -1.7374,E1 24.959,E2 194.5857} C_DIS
LIN {X -23.0193,Y -99.4634,Z 105,A -106.7505,B 24.9432,C -1.7415,E1 24.9653,E2 192.2719} C_DIS
LIN {X -19.7275,Y -100.1691,Z 105,A -104.7583,B 24.943,C -1.7446,E1 24.9708,E2 190.2701} C_DIS
LIN {X -16.3203,Y -100.7808,Z 105,A -102.8088,B 24.943,C -1.7443,E1 24.9762,E2 188.3195} C_DIS
LIN {X -12.942,Y -101.2689,Z 105,A -100.8828,B 24.943,C -1.7443,E1 24.9815,E2 186.392} C_DIS
LIN {X -9.1643,Y -101.6804,Z 105,A -98.7226,B 24.943,C -1.7451,E1 24.9875,E2 184.2286} C_DIS
LIN {X -5.2686,Y -101.957,Z 105,A -96.7307,B 24.9434,C -1.7375,E1 24.993,E2 182.2541} C_DIS
LIN {X -2.424,Y -102.065,Z 105,A -94.9253,B 24.9429,C -1.7457,E1 24.9981,E2 180.4289} C_DIS
LIN {X 0.721,Y -102.0888,Z 105,A -93.969,B 24.9449,C -1.715,E1 25.0006,E2 179.5454} C_DIS
Enddeposition()
LIN {X 0.721,Y -102.0888,Z 105,A -93.969,B 24.9449,C -1.715,E1 25.0006,E2 179.5454} C_DIS
Startdeposition()
$VEL.CP = VEL_PRINT
LIN {X -0.7043,Y -101.1093,Z 105,A -94.9326,B 24.9442,C -1.7262,E1 24.998,E2 180.4826} C_DIS
LIN {X -3.7243,Y -101.045,Z 105,A -96.5555,B 24.944,C -1.7292,E1 24.9934,E2 182.0985} C_DIS
LIN {X -6.1969,Y -100.9235,Z 105,A -97.9586,B 24.944,C -1.7292,E1 24.9895,E2 183.5021} C_DIS
LIN {X -8.6794,Y -100.7404,Z 105,A -99.3689,B 24.944,C -1.7292,E1 24.9856,E2 184.913} C_DIS
LIN {X -11.6014,Y -100.4441,Z 105,A -101.132,B 24.9442,C -1.7257,E1 24.9807,E2 186.6853} C_DIS
LIN {X -14.8383,Y -100.019,Z 105,A -102.8849,B 24.9439,C -1.7297,E1 24.9759,E2 188.4302} C_DIS
LIN {X -18.1129,Y -99.4764,Z 105,A -104.7812,B 24.9439,C -1.7297,E1 24.9706,E2 190.3282} C_DIS
LIN {X -20.7618,Y -98.9582,Z 105,A -106.4868,B 24.9443,C -1.7239,E1 24.9659,E2 192.0498} C_DIS
LIN {X -24.3402,Y -98.1391,Z 105,A -108.5728,B 24.9443,C -1.7248,E1 24.9603,E2 194.1364} C_DIS
LIN {X -27.7977,Y -97.2159,Z 105,A -110.4637,B 24.9438,C -1.7311,E1 24.9552,E2 196.0153} C_DIS
LIN {X -30.5421,Y -96.3906,Z 105,A -112.0359,B 24.9436,C -1.7341,E1 24.951,E2 197.583} C_DIS
LIN {X -32.8885,Y -95.6154,Z 105,A -113.4401,B 24.9436,C -1.7351,E1 24.9473,E2 198.9875} C_DIS
LIN {X -35.2413,Y -94.7734,Z 105,A -114.8589,B 24.9436,C -1.7363,E1 24.9436,E2 200.4064} C_DIS
LIN {X -38.3318,Y -93.5645,Z 105,A -116.7951,B 24.9436,C -1.7361,E1 24.9385,E2 202.3472} C_DIS
LIN {X -40.9755,Y -92.4391,Z 105,A -118.3769,B 24.9433,C -1.7395,E1 24.9345,E2 203.9246} C_DIS
LIN {X -43.2274,Y -91.4076,Z 105,A -119.7841,B 24.9432,C -1.741,E1 24.9309,E2 205.3318} C_DIS
LIN {X -45.4533,Y -90.3214,Z 105,A -121.3998,B 24.9436,C -1.7351,E1 24.9269,E2 206.9659} C_DIS
LIN {X -48.4194,Y -88.7648,Z 105,A -123.3008,B 24.9434,C -1.7375,E1 24.9222,E2 208.8664} C_DIS
LIN {X -51.446,Y -87.0454,Z 105,A -125.1249,B 24.9429,C -1.7457,E1 24.9178,E2 210.6766} C_DIS
LIN {X -53.7612,Y -85.6351,Z 105,A -126.6145,B 24.9426,C -1.7496,E1 24.9143,E2 212.1615} C_DIS
LIN {X -56.1738,Y -84.0742,Z 105,A -128.2481,B 24.9425,C -1.752,E1 24.9105,E2 213.7948} C_DIS
LIN {X -59.2246,Y -81.9537,Z 105,A -130.3596,B 24.9423,C -1.7553,E1 24.9056,E2 215.9057} C_DIS
LIN {X -62.2138,Y -79.7083,Z 105,A -132.6509,B 24.9424,C -1.7529,E1 24.9005,E2 218.2109} C_DIS
LIN {X -64.6224,Y -77.7658,Z 105,A -134.2935,B 24.9419,C -1.7602,E1 24.897,E2 219.8425} C_DIS
LIN {X -67.1217,Y -75.6204,Z 105,A -136.2657,B 24.9419,C -1.76,E1 24.8928,E2 221.8227} C_DIS
LIN {X -69.4232,Y -73.5122,Z 105,A -138.0436,B 24.9417,C -1.7633,E1 24.8892,E2 223.6001} C_DIS
LIN {X -71.9363,Y -71.0546,Z 105,A -139.9452,B 24.9412,C -1.7707,E1 24.8854,E2 225.4922} C_DIS
LIN {X -74.2124,Y -68.6752,Z 105,A -141.9145,B 24.9412,C -1.7712,E1 24.8817,E2 227.4689} C_DIS
LIN {X -76.4248,Y -66.2043,Z 105,A -143.8486,B 24.941,C -1.7735,E1 24.8781,E2 229.4061} C_DIS
LIN {X -78.5791,Y -63.631,Z 105,A -145.6747,B 24.9406,C -1.7806,E1 24.8749,E2 231.2236} C_DIS
LIN {X -81.0101,Y -60.5064,Z 105,A -147.7042,B 24.9397,C -1.7935,E1 24.8714,E2 233.2322} C_DIS
LIN {X -82.5146,Y -58.4384,Z 105,A -149.2882,B 24.9397,C -1.7924,E1 24.8688,E2 234.8265} C_DIS
LIN {X -84.0777,Y -56.1685,Z 105,A -150.8549,B 24.9395,C -1.7962,E1 24.8664,E2 236.3919} C_DIS
LIN {X -85.4284,Y -54.0921,Z 105,A -152.2701,B 24.9393,C -1.7994,E1 24.8642,E2 237.8066} C_DIS
LIN {X -86.7279,Y -51.9831,Z 105,A -153.6829,B 24.9391,C -1.8028,E1 24.8622,E2 239.2186} C_DIS
LIN {X -88.3865,Y -49.1065,Z 105,A -155.6291,B 24.9389,C -1.8057,E1 24.8595,E2 241.1681} C_DIS
LIN {X -90.1344,Y -45.8195,Z 105,A -157.7486,B 24.9385,C -1.8112,E1 24.8568,E2 243.2858} C_DIS
LIN {X -91.3987,Y -43.2461,Z 105,A -159.514,B 24.9385,C -1.8109,E1 24.8546,E2 245.0614} C_DIS
LIN {X -92.7787,Y -40.1965,Z 105,A -161.2413,B 24.9378,C -1.8221,E1 24.8527,E2 246.7715} C_DIS
LIN {X -93.8849,Y -37.5445,Z 105,A -162.8798,B 24.9375,C -1.8265,E1 24.8509,E2 248.4087} C_DIS
LIN {X -95.0651,Y -34.4421,Z 105,A -164.7382,B 24.937,C -1.8328,E1 24.8491,E2 250.2624} C_DIS
LIN {X -95.8883,Y -32.0791,Z 105,A -166.2001,B 24.9368,C -1.8355,E1 24.8478,E2 251.7263} C_DIS
LIN {X -96.6445,Y -29.7234,Z 105,A -167.6114,B 24.9366,C -1.8394,E1 24.8466,E2 253.1363} C_DIS
LIN {X -97.4509,Y -26.9683,Z 105,A -169.2496,B 24.9363,C -1.844,E1 24.8454,E2 254.7732} C_DIS
LIN {X -98.3804,Y -23.3504,Z 105,A -171.3737,B 24.9358,C -1.8502,E1 24.8439,E2 256.8948} C_DIS
LIN {X -99.1688,Y -19.7357,Z 105,A -173.4891,B 24.9354,C -1.8561,E1 24.8427,E2 259.0086} C_DIS
LIN {X -99.6857,Y -16.9232,Z 105,A -175.2045,B 24.9353,C -1.858,E1 24.8419,E2 260.7297} C_DIS
LIN {X -100.1388,Y -13.9951,Z 105,A -176.8644,B 24.9349,C -1.8639,E1 24.8412,E2 262.3854} C_DIS
LIN {X -100.4976,Y -11.1442,Z 105,A -178.4529,B 24.9344,C -1.8704,E1 24.8407,E2 263.9679} C_DIS
LIN {X -100.8076,Y -7.8394,Z 105,A 179.6016,B 24.9341,C -1.8743,E1 24.8402,E2 265.9159} C_DIS
LIN {X -101.0195,Y -4.3179,Z 105,A 177.5358,B 24.9339,C -1.8784,E1 24.8399,E2 267.9842} C_DIS
LIN {X -101.109,Y -0.7817,Z 105,A 175.5363,B 24.9334,C -1.8851,E1 24.8398,E2 269.9799} C_DIS
LIN {X -101.0833,Y 2.4767,Z 105,A 173.7617,B 24.9328,C -1.8934,E1 24.8398,E2 271.7453} C_DIS
LIN {X -100.9705,Y 5.3484,Z 105,A 172.0267,B 24.9327,C -1.8951,E1 24.8401,E2 273.4867} C_DIS
LIN {X -100.7413,Y 8.669,Z 105,A 170.0151,B 24.9325,C -1.897,E1 24.8405,E2 275.5059} C_DIS
LIN {X -100.3856,Y 12.1013,Z 105,A 168.0447,B 24.9321,C -1.9028,E1 24.8411,E2 277.4743} C_DIS
LIN {X -99.8908,Y 15.6671,Z 105,A 166.1928,B 24.9312,C -1.9157,E1 24.8419,E2 279.3064} C_DIS
LIN {X -99.4738,Y 18.1271,Z 105,A 164.7263,B 24.931,C -1.9184,E1 24.8426,E2 280.775} C_DIS
LIN {X -99.0049,Y 20.5343,Z 105,A 163.311,B 24.9307,C -1.922,E1 24.8434,E2 282.1902} C_DIS
LIN {X -98.3743,Y 23.3764,Z 105,A 161.7202,B 24.9302,C -1.9292,E1 24.8444,E2 283.7731} C_DIS
LIN {X -97.4498,Y 26.9723,Z 105,A 159.5964,B 24.9298,C -1.9352,E1 24.8459,E2 285.895} C_DIS
LIN {X -96.7603,Y 29.3499,Z 105,A 158.1818,B 24.9295,C -1.9392,E1 24.847,E2 287.3081} C_DIS
LIN {X -96.0127,Y 31.7098,Z 105,A 156.7694,B 24.9292,C -1.9433,E1 24.8482,E2 288.719} C_DIS
LIN {X -95.3389,Y 33.6766,Z 105,A 155.5315,B 24.9291,C -1.945,E1 24.8493,E2 289.9599} C_DIS
LIN {X -94.0319,Y 37.1703,Z 105,A 153.4408,B 24.9285,C -1.9523,E1 24.8514,E2 292.0449} C_DIS
LIN {X -92.7581,Y 40.2436,Z 105,A 151.4501,B 24.9284,C -1.9545,E1 24.8536,E2 294.0414} C_DIS
LIN {X -91.4028,Y 43.2376,Z 105,A 149.6859,B 24.9277,C -1.9634,E1 24.8556,E2 295.7941} C_DIS
LIN {X -90.5005,Y 45.0919,Z 105,A 148.4474,B 24.9277,C -1.9645,E1 24.8572,E2 297.0365} C_DIS
LIN {X -89.1715,Y 47.6697,Z 105,A 146.8555,B 24.9272,C -1.9711,E1 24.8592,E2 298.6213} C_DIS
LIN {X -87.7816,Y 50.18,Z 105,A 145.1299,B 24.9271,C -1.9724,E1 24.8616,E2 300.3527} C_DIS
LIN {X -86.1655,Y 52.9084,Z 105,A 143.3994,B 24.9265,C -1.9798,E1 24.8641,E2 302.0744} C_DIS
LIN {X -84.4609,Y 55.5873,Z 105,A 141.5111,B 24.9264,C -1.9819,E1 24.8669,E2 303.9673} C_DIS
LIN {X -82.4371,Y 58.547,Z 105,A 139.4463,B 24.926,C -1.9864,E1 24.8702,E2 306.0316} C_DIS
LIN {X -80.7041,Y 60.9137,Z 105,A 137.8296,B 24.9256,C -1.9924,E1 24.8729,E2 307.6417} C_DIS
LIN {X -78.6765,Y 63.5109,Z 105,A 135.9441,B 24.9252,C -1.9967,E1 24.8762,E2 309.5257} C_DIS
LIN {X -76.8393,Y 65.7217,Z 105,A 134.3083,B 24.9249,C -2.0007,E1 24.8791,E2 311.1596} C_DIS
LIN {X -74.5702,Y 68.2853,Z 105,A 132.3387,B 24.9247,C -2.0046,E1 24.8828,E2 313.1287} C_DIS
LIN {X -72.3682,Y 70.6173,Z 105,A 130.4227,B 24.9246,C -2.0057,E1 24.8865,E2 315.0504} C_DIS
LIN {X -70.1701,Y 72.7993,Z 105,A 128.7397,B 24.9241,C -2.0124,E1 24.8898,E2 316.7245} C_DIS
LIN {X -67.7618,Y 75.0473,Z 105,A 126.809,B 24.9239,C -2.0145,E1 24.8938,E2 318.6579} C_DIS
LIN {X -65.2476,Y 77.2432,Z 105,A 124.9401,B 24.9235,C -2.0196,E1 24.8978,E2 320.5221} C_DIS
LIN {X -62.6956,Y 79.3275,Z 105,A 123.0863,B 24.9232,C -2.0241,E1 24.9018,E2 322.372} C_DIS
LIN {X -60.239,Y 81.211,Z 105,A 121.4062,B 24.9227,C -2.0303,E1 24.9055,E2 324.0433} C_DIS
LIN {X -58.231,Y 82.6626,Z 105,A 119.8197,B 24.923,C -2.0268,E1 24.9092,E2 325.6437} C_DIS
LIN {X -55.4319,Y 84.5633,Z 105,A 118.0119,B 24.9224,C -2.0344,E1 24.9133,E2 327.4394} C_DIS
LIN {X -53.0177,Y 86.0991,Z 105,A 116.4458,B 24.922,C -2.0394,E1 24.917,E2 328.9986} C_DIS
LIN {X -50.1725,Y 87.7859,Z 105,A 114.5615,B 24.9218,C -2.0424,E1 24.9216,E2 330.8814} C_DIS
LIN {X -47.6662,Y 89.1734,Z 105,A 112.9314,B 24.9216,C -2.0449,E1 24.9256,E2 332.5101} C_DIS
LIN {X -44.3681,Y 90.8593,Z 105,A 110.8298,B 24.9213,C -2.0482,E1 24.9308,E2 334.6095} C_DIS
LIN {X -40.9707,Y 92.4411,Z 105,A 108.6965,B 24.9211,C -2.0511,E1 24.9362,E2 336.7411} C_DIS
LIN {X -37.5468,Y 93.884,Z 105,A 106.5819,B 24.9209,C -2.0538,E1 24.9416,E2 338.8542} C_DIS
LIN {X -35.2236,Y 94.78,Z 105,A 105.0038,B 24.9212,C -2.0497,E1 24.9458,E2 340.4453} C_DIS
LIN {X -32.0734,Y 95.8903,Z 105,A 103.2696,B 24.9206,C -2.0577,E1 24.9503,E2 342.1638} C_DIS
LIN {X -29.7203,Y 96.6454,Z 105,A 101.8657,B 24.9205,C -2.0592,E1 24.9541,E2 343.5667} C_DIS
LIN {X -26.968,Y 97.451,Z 105,A 100.236,B 24.9204,C -2.0607,E1 24.9585,E2 345.1953} C_DIS
LIN {X -24.5773,Y 98.0812,Z 105,A 98.832,B 24.9203,C -2.062,E1 24.9622,E2 346.5983} C_DIS
LIN {X -21.3518,Y 98.8318,Z 105,A 96.8992,B 24.9203,C -2.0617,E1 24.9675,E2 348.5342} C_DIS
LIN {X -18.1173,Y 99.4756,Z 105,A 95.0027,B 24.9203,C -2.0622,E1 24.9727,E2 350.4317} C_DIS
LIN {X -14.8266,Y 100.0206,Z 105,A 93.1917,B 24.9199,C -2.0664,E1 24.9777,E2 352.2344} C_DIS
LIN {X -12.3721,Y 100.3538,Z 105,A 91.7822,B 24.9199,C -2.067,E1 24.9816,E2 353.6435} C_DIS
LIN {X -10.3044,Y 100.5856,Z 105,A 90.5506,B 24.9199,C -2.0658,E1 24.985,E2 354.8787} C_DIS
LIN {X -6.9214,Y 100.8746,Z 105,A 88.5931,B 24.92,C -2.0654,E1 24.9905,E2 356.8379} C_DIS
LIN {X -3.71,Y 101.0455,Z 105,A 86.8569,B 24.9197,C -2.0691,E1 24.9953,E2 358.5657} C_DIS
LIN {X 0.0038,Y 101.1136,Z 105,A 84.7468,B 24.9197,C -2.0694,E1 25.0012,E2 360.6751} C_DIS
LIN {X 2.4802,Y 101.0832,Z 105,A 83.341,B 24.9197,C -2.0695,E1 25.0051,E2 362.0805} C_DIS
LIN {X 4.9551,Y 100.9921,Z 105,A 81.7477,B 24.9202,C -2.0626,E1 25.0096,E2 363.6897} C_DIS
LIN {X 8.1682,Y 100.7813,Z 105,A 80.0333,B 24.9199,C -2.0666,E1 25.0143,E2 365.3938} C_DIS
LIN {X 11.148,Y 100.4972,Z 105,A 78.4187,B 24.9197,C -2.0694,E1 25.0188,E2 367.0008} C_DIS
LIN {X 14.8328,Y 100.0198,Z 105,A 76.3135,B 24.9197,C -2.0689,E1 25.0246,E2 369.1053} C_DIS
LIN {X 17.202,Y 99.6391,Z 105,A 74.7526,B 24.9203,C -2.061,E1 25.029,E2 370.6835} C_DIS
LIN {X 20.6269,Y 98.9859,Z 105,A 72.9661,B 24.9199,C -2.0672,E1 25.0338,E2 372.4531} C_DIS
LIN {X 23.1358,Y 98.43,Z 105,A 71.5413,B 24.9199,C -2.0676,E1 25.0377,E2 373.875} C_DIS
LIN {X 25.4004,Y 97.8696,Z 105,A 70.1547,B 24.9201,C -2.0644,E1 25.0415,E2 375.2672} C_DIS
LIN {X 27.7843,Y 97.2197,Z 105,A 68.7582,B 24.9201,C -2.0636,E1 25.0452,E2 376.6633} C_DIS
LIN {X 30.2919,Y 96.4682,Z 105,A 67.2962,B 24.9201,C -2.0632,E1 25.0491,E2 378.1235} C_DIS
LIN {X 32.9043,Y 95.6099,Z 105,A 65.7769,B 24.9201,C -2.0634,E1 25.0531,E2 379.6394} C_DIS
LIN {X 35.2359,Y 94.7755,Z 105,A 64.3738,B 24.9203,C -2.0621,E1 25.0568,E2 381.0427} C_DIS
LIN {X 38.3265,Y 93.5666,Z 105,A 62.444,B 24.9206,C -2.0583,E1 25.0618,E2 382.977} C_DIS
LIN {X 40.97,Y 92.4414,Z 105,A 60.8711,B 24.9206,C -2.0586,E1 25.0659,E2 384.5455} C_DIS
LIN {X 43.2344,Y 91.4043,Z 105,A 59.4636,B 24.9206,C -2.0571,E1 25.0694,E2 385.953} C_DIS
LIN {X 46.3355,Y 89.8707,Z 105,A 57.4811,B 24.9209,C -2.0538,E1 25.0744,E2 387.938} C_DIS
LIN {X 48.4054,Y 88.7725,Z 105,A 55.9746,B 24.9216,C -2.0451,E1 25.0781,E2 389.4606} C_DIS
LIN {X 51.5664,Y 86.9742,Z 105,A 54.1123,B 24.9212,C -2.0498,E1 25.0826,E2 391.3063} C_DIS
LIN {X 53.7564,Y 85.6381,Z 105,A 52.6801,B 24.9213,C -2.0484,E1 25.086,E2 392.7372} C_DIS
LIN {X 56.1683,Y 84.0778,Z 105,A 51.0577,B 24.9215,C -2.046,E1 25.0898,E2 394.3601} C_DIS
LIN {X 58.6726,Y 82.3475,Z 105,A 49.2695,B 24.9219,C -2.0406,E1 25.0939,E2 396.1546} C_DIS
LIN {X 60.912,Y 80.7054,Z 105,A 47.7226,B 24.922,C -2.0389,E1 25.0973,E2 397.7002} C_DIS
LIN {X 63.5055,Y 78.6808,Z 105,A 45.8541,B 24.9223,C -2.0353,E1 25.1014,E2 399.5702} C_DIS
LIN {X 65.6683,Y 76.8848,Z 105,A 44.2436,B 24.9226,C -2.0315,E1 25.1049,E2 401.1833} C_DIS
LIN {X 68.3701,Y 74.4924,Z 105,A 42.2491,B 24.9228,C -2.0294,E1 25.109,E2 403.1749} C_DIS
LIN {X 70.617,Y 72.3686,Z 105,A 40.3867,B 24.9234,C -2.0214,E1 25.1128,E2 405.0485} C_DIS
LIN {X 72.7947,Y 70.1749,Z 105,A 38.7195,B 24.9234,C -2.0209,E1 25.116,E2 406.7096} C_DIS
LIN {X 75.0543,Y 67.754,Z 105,A 36.8007,B 24.9239,C -2.015,E1 25.1197,E2 408.6339} C_DIS
LIN {X 77.2473,Y 65.2429,Z 105,A 34.9537,B 24.9241,C -2.0123,E1 25.123,E2 410.4789} C_DIS
LIN {X 79.3272,Y 62.696,Z 105,A 33.1225,B 24.9243,C -2.0092,E1 25.1262,E2 412.3091} C_DIS
LIN {X 81.2152,Y 60.2333,Z 105,A 31.2444,B 24.925,C -2.0001,E1 25.1294,E2 414.1996} C_DIS
LIN {X 83.2598,Y 57.3722,Z 105,A 29.4527,B 24.9248,C -2.003,E1 25.1322,E2 415.9756} C_DIS
LIN {X 84.541,Y 55.4658,Z 105,A 27.9732,B 24.9256,C -1.9926,E1 25.1345,E2 417.4723} C_DIS
LIN {X 86.4588,Y 52.4258,Z 105,A 26.1178,B 24.9254,C -1.9945,E1 25.1373,E2 419.314} C_DIS
LIN {X 87.9894,Y 49.8177,Z 105,A 24.2497,B 24.9262,C -1.9837,E1 25.1399,E2 421.1979} C_DIS
LIN {X 89.5671,Y 46.9188,Z 105,A 22.5401,B 24.9262,C -1.985,E1 25.1421,E2 422.8954} C_DIS
LIN {X 91.0823,Y 43.9046,Z 105,A 20.6026,B 24.9266,C -1.9786,E1 25.1445,E2 424.8376} C_DIS
LIN {X 92.2012,Y 41.5033,Z 105,A 19.1586,B 24.9267,C -1.9766,E1 25.1462,E2 426.2786} C_DIS
LIN {X 93.2634,Y 39.0587,Z 105,A 17.6476,B 24.9271,C -1.9722,E1 25.1478,E2 427.7916} C_DIS
LIN {X 94.6682,Y 35.5193,Z 105,A 15.3472,B 24.928,C -1.9601,E1 25.1502,E2 430.1077} C_DIS
LIN {X 95.8944,Y 32.0611,Z 105,A 13.4887,B 24.9278,C -1.9628,E1 25.1519,E2 431.9494} C_DIS
LIN {X 96.6451,Y 29.7213,Z 105,A 12.1052,B 24.9281,C -1.959,E1 25.153,E2 433.3341} C_DIS
LIN {X 97.4466,Y 26.9834,Z 105,A 10.5012,B 24.9284,C -1.9545,E1 25.1543,E2 434.9394} C_DIS
LIN {X 98.0836,Y 24.5678,Z 105,A 8.9008,B 24.9292,C -1.9427,E1 25.1554,E2 436.5585} C_DIS
LIN {X 98.8357,Y 21.3337,Z 105,A 7.1723,B 24.9292,C -1.9431,E1 25.1564,E2 438.276} C_DIS
LIN {X 99.3287,Y 18.9062,Z 105,A 5.6213,B 24.93,C -1.9327,E1 25.1573,E2 439.8424} C_DIS
LIN {X 99.9475,Y 15.3006,Z 105,A 3.7554,B 24.9298,C -1.9346,E1 25.1581,E2 441.693} C_DIS
LIN {X 100.3531,Y 12.378,Z 105,A 2.1086,B 24.9301,C -1.9303,E1 25.1587,E2 443.3403} C_DIS
LIN {X 100.7037,Y 9.0776,Z 105,A 0.2413,B 24.9305,C -1.9248,E1 25.1592,E2 445.2093} C_DIS
LIN {X 100.9233,Y 6.2017,Z 105,A -1.3819,B 24.9309,C -1.92,E1 25.1595,E2 446.8343} C_DIS
LIN {X 101.0454,Y 3.7132,Z 105,A -2.7823,B 24.9312,C -1.9159,E1 25.1597,E2 448.236} C_DIS
LIN {X 101.109,Y 0.7821,Z 105,A -4.5168,B 24.9318,C -1.9076,E1 25.1597,E2 449.9798} C_DIS
LIN {X 101.0834,Y -2.4723,Z 105,A -6.2722,B 24.9319,C -1.9052,E1 25.1597,E2 451.7303} C_DIS
LIN {X 101.0084,Y -4.5761,Z 105,A -7.5009,B 24.9323,C -1.8999,E1 25.1596,E2 452.9642} C_DIS
LIN {X 100.8661,Y -7.0479,Z 105,A -8.8927,B 24.9326,C -1.8959,E1 25.1593,E2 454.3573} C_DIS
LIN {X 100.6268,Y -9.9104,Z 105,A -10.4593,B 24.9328,C -1.893,E1 25.1589,E2 455.9213} C_DIS
LIN {X 100.4,Y -11.978,Z 105,A -11.833,B 24.9337,C -1.8813,E1 25.1585,E2 457.3145} C_DIS
LIN {X 99.9188,Y -15.4859,Z 105,A -13.7201,B 24.9337,C -1.8797,E1 25.1577,E2 459.1943} C_DIS
LIN {X 99.2959,Y -19.0763,Z 105,A -15.7527,B 24.9341,C -1.8744,E1 25.1567,E2 461.2276} C_DIS
LIN {X 98.552,Y -22.6077,Z 105,A -17.806,B 24.9346,C -1.8675,E1 25.1555,E2 463.2852} C_DIS
LIN {X 97.8655,Y -25.4165,Z 105,A -19.3812,B 24.9348,C -1.8648,E1 25.1544,E2 464.8576} C_DIS
LIN {X 97.219,Y -27.7868,Z 105,A -20.7613,B 24.9351,C -1.8609,E1 25.1534,E2 466.239} C_DIS
LIN {X 96.4607,Y -30.3161,Z 105,A -22.2249,B 24.9353,C -1.8575,E1 25.1522,E2 467.7023} C_DIS
LIN {X 95.6114,Y -32.9002,Z 105,A -23.7279,B 24.9356,C -1.8542,E1 25.1508,E2 469.2046} C_DIS
LIN {X 94.5753,Y -35.7646,Z 105,A -25.5091,B 24.9361,C -1.8466,E1 25.1491,E2 470.9937} C_DIS
LIN {X 93.5646,Y -38.3314,Z 105,A -27.0472,B 24.9363,C -1.8428,E1 25.1475,E2 472.5323} C_DIS
LIN {X 92.44,Y -40.9733,Z 105,A -28.6139,B 24.9365,C -1.8403,E1 25.1458,E2 474.0964} C_DIS
LIN {X 90.8735,Y -44.3392,Z 105,A -30.7015,B 24.9369,C -1.8346,E1 25.1433,E2 476.1862} C_DIS
LIN {X 89.7612,Y -46.5496,Z 105,A -32.2661,B 24.9376,C -1.8239,E1 25.1413,E2 477.7678} C_DIS
LIN {X 88.1026,Y -49.615,Z 105,A -34.0879,B 24.9376,C -1.8243,E1 25.1388,E2 479.5791} C_DIS
LIN {X 86.7241,Y -51.9893,Z 105,A -35.6023,B 24.9378,C -1.8214,E1 25.1367,E2 481.0925} C_DIS
LIN {X 84.9697,Y -54.8068,Z 105,A -37.5249,B 24.9383,C -1.8144,E1 25.1338,E2 483.022} C_DIS
LIN {X 83.3789,Y -57.2008,Z 105,A -39.2867,B 24.939,C -1.8044,E1 25.131,E2 484.7986} C_DIS
LIN {X 81.4408,Y -59.9253,Z 105,A -40.9773,B 24.9388,C -1.8075,E1 25.1283,E2 486.4738} C_DIS
LIN {X 79.7076,Y -62.2147,Z 105,A -42.7558,B 24.9395,C -1.7969,E1 25.1252,E2 488.2687} C_DIS
LIN {X 77.7649,Y -64.6236,Z 105,A -44.3827,B 24.9395,C -1.7974,E1 25.1224,E2 489.8869} C_DIS
LIN {X 75.7432,Y -66.9845,Z 105,A -46.305,B 24.9402,C -1.7864,E1 25.1188,E2 491.8267} C_DIS
LIN {X 73.5122,Y -69.4233,Z 105,A -48.0102,B 24.9401,C -1.7884,E1 25.1156,E2 493.5196} C_DIS
LIN {X 71.1954,Y -71.7972,Z 105,A -49.8802,B 24.9403,C -1.7842,E1 25.1119,E2 495.3917} C_DIS
LIN {X 68.9655,Y -73.9427,Z 105,A -51.5855,B 24.9405,C -1.7819,E1 25.1085,E2 497.0953} C_DIS
LIN {X 66.5028,Y -76.164,Z 105,A -53.517,B 24.9409,C -1.7755,E1 25.1044,E2 499.0342} C_DIS
LIN {X 63.9867,Y -78.2909,Z 105,A -55.4304,B 24.9413,C -1.7694,E1 25.1003,E2 500.9546} C_DIS
LIN {X 61.3837,Y -80.348,Z 105,A -57.1805,B 24.9413,C -1.7705,E1 25.0964,E2 502.6956} C_DIS
LIN {X 59.2384,Y -81.9437,Z 105,A -58.6728,B 24.9413,C -1.7682,E1 25.0931,E2 504.188} C_DIS
LIN {X 57.1979,Y -83.3808,Z 105,A -60.0815,B 24.9416,C -1.7656,E1 25.0899,E2 505.5983} C_DIS
LIN {X 55.4692,Y -84.5387,Z 105,A -61.3063,B 24.9418,C -1.7615,E1 25.087,E2 506.8287} C_DIS
LIN {X 53.0444,Y -86.0829,Z 105,A -62.8789,B 24.9419,C -1.7605,E1 25.0833,E2 508.3984} C_DIS
LIN {X 50.1895,Y -87.7761,Z 105,A -64.752,B 24.9421,C -1.7574,E1 25.0788,E2 510.2732} C_DIS
LIN {X 47.676,Y -89.1681,Z 105,A -66.3744,B 24.9423,C -1.7548,E1 25.0748,E2 511.8972} C_DIS
LIN {X 45.0787,Y -90.5071,Z 105,A -68.1343,B 24.9427,C -1.748,E1 25.0704,E2 513.6683} C_DIS
LIN {X 42.4486,Y -91.7701,Z 105,A -69.7246,B 24.9427,C -1.7478,E1 25.0664,E2 515.255} C_DIS
LIN {X 39.0526,Y -93.2659,Z 105,A -71.818,B 24.9429,C -1.745,E1 25.061,E2 517.3499} C_DIS
LIN {X 36.3899,Y -94.3385,Z 105,A -73.3895,B 24.9429,C -1.7449,E1 25.0569,E2 518.9183} C_DIS
LIN {X 32.8818,Y -95.6177,Z 105,A -75.4932,B 24.9431,C -1.7426,E1 25.0514,E2 521.0231} C_DIS
LIN {X 29.6687,Y -96.6615,Z 105,A -77.6142,B 24.9438,C -1.7323,E1 25.0457,E2 523.1644} C_DIS
LIN {X 26.1359,Y -97.6758,Z 105,A -79.5341,B 24.9435,C -1.7363,E1 25.0406,E2 525.0716} C_DIS
LIN {X 23.373,Y -98.3751,Z 105,A -81.096,B 24.9435,C -1.7367,E1 25.0363,E2 526.6304} C_DIS
LIN {X 19.7199,Y -99.172,Z 105,A -83.21,B 24.9435,C -1.735,E1 25.0306,E2 528.7456} C_DIS
LIN {X 17.2846,Y -99.6253,Z 105,A -84.6134,B 24.9437,C -1.7339,E1 25.0267,E2 530.1502} C_DIS
LIN {X 14.8389,Y -100.0189,Z 105,A -86.1737,B 24.9441,C -1.7269,E1 25.0223,E2 531.7256} C_DIS
LIN {X 11.5914,Y -100.4453,Z 105,A -87.8808,B 24.9438,C -1.7314,E1 25.0176,E2 533.4206} C_DIS
LIN {X 9.0633,Y -100.705,Z 105,A -89.3076,B 24.9438,C -1.7312,E1 25.0137,E2 534.8471} C_DIS
LIN {X 6.1989,Y -100.9234,Z 105,A -91.115,B 24.9443,C -1.7236,E1 25.0086,E2 536.6717} C_DIS
LIN {X 2.8581,Y -101.0716,Z 105,A -93.0348,B 24.9444,C -1.722,E1 25.0032,E2 538.5948} C_DIS
LIN {X 2.8581,Y -101.0716,Z 105,A -93.0348,B 24.9444,C -1.722,E1 25.0032,E2 538.5948} C_DIS
Enddeposition()
LIN {X 0.7495,Y -107.8071,Z 106,A -93.5299,B 24.9496,C -1.6393,E1 25.0013,E2 539.2858} C_DIS
Startdeposition()
$VEL.CP = VEL_PRINT
LIN {X 3.1194,Y -107.7647,Z 106,A -92.1069,B 24.9492,C -1.6464,E1 25.0053,E2 537.8464} C_DIS
LIN {X 5.7631,Y -107.6557,Z 106,A -90.503,B 24.9487,C -1.655,E1 25.0099,E2 536.2224} C_DIS
LIN {X 8.0539,Y -107.5097,Z 106,A -89.3437,B 24.9487,C -1.6531,E1 25.0131,E2 535.0683} C_DIS
LIN {X 11.0386,Y -107.2432,Z 106,A -87.9229,B 24.9492,C -1.6468,E1 25.017,E2 533.6631} C_DIS
LIN {X 13.1973,Y -107.0009,Z 106,A -86.3716,B 24.9481,C -1.664,E1 25.0214,E2 532.0724} C_DIS
LIN {X 17.1268,Y -106.4426,Z 106,A -84.2656,B 24.9481,C -1.6654,E1 25.0272,E2 529.9651} C_DIS
LIN {X 20.199,Y -105.9007,Z 106,A -82.7792,B 24.9484,C -1.6596,E1 25.0312,E2 528.4941} C_DIS
LIN {X 23.0803,Y -105.3102,Z 106,A -81.1401,B 24.9481,C -1.6642,E1 25.0357,E2 526.8462} C_DIS
LIN {X 26.1961,Y -104.5807,Z 106,A -79.3455,B 24.9478,C -1.6698,E1 25.0406,E2 525.0409} C_DIS
LIN {X 28.7548,Y -103.9063,Z 106,A -78.1189,B 24.9481,C -1.6637,E1 25.0439,E2 523.8307} C_DIS
LIN {X 31.7486,Y -103.029,Z 106,A -76.4651,B 24.9481,C -1.6655,E1 25.0483,E2 522.1755} C_DIS
LIN {X 35.0723,Y -101.9475,Z 106,A -74.4438,B 24.9474,C -1.6747,E1 25.0537,E2 520.1364} C_DIS
LIN {X 38.275,Y -100.7867,Z 106,A -72.7262,B 24.9475,C -1.6732,E1 25.0582,E2 518.4259} C_DIS
LIN {X 41.6943,Y -99.421,Z 106,A -70.8564,B 24.9475,C -1.6723,E1 25.063,E2 516.5625} C_DIS
LIN {X 44.896,Y -98.0189,Z 106,A -69.0049,B 24.9475,C -1.6749,E1 25.0677,E2 514.7095} C_DIS
LIN {X 47.7124,Y -96.6772,Z 106,A -67.3527,B 24.9473,C -1.6773,E1 25.0719,E2 513.0558} C_DIS
LIN {X 50.0706,Y -95.4772,Z 106,A -65.9516,B 24.9471,C -1.6795,E1 25.0754,E2 511.6535} C_DIS
LIN {X 53.1402,Y -93.8055,Z 106,A -64.0722,B 24.9469,C -1.6837,E1 25.08,E2 509.7697} C_DIS
LIN {X 55.4263,Y -92.4732,Z 106,A -62.6724,B 24.9467,C -1.686,E1 25.0834,E2 508.3687} C_DIS
LIN {X 58.0777,Y -90.8292,Z 106,A -61.2778,B 24.9472,C -1.6779,E1 25.0866,E2 506.9976} C_DIS
LIN {X 60.2892,Y -89.3765,Z 106,A -59.649,B 24.9465,C -1.6903,E1 25.0904,E2 505.3451} C_DIS
LIN {X 63.1559,Y -87.3768,Z 106,A -57.7994,B 24.9462,C -1.6937,E1 25.0947,E2 503.4938} C_DIS
LIN {X 65.2812,Y -85.8005,Z 106,A -56.3996,B 24.9461,C -1.6964,E1 25.0978,E2 502.0927} C_DIS
LIN {X 67.3672,Y -84.1726,Z 106,A -55.0001,B 24.9459,C -1.6992,E1 25.1009,E2 500.6918} C_DIS
LIN {X 69.7732,Y -82.1867,Z 106,A -53.5785,B 24.9463,C -1.6928,E1 25.1039,E2 499.2909} C_DIS
LIN {X 71.7691,Y -80.4497,Z 106,A -51.9508,B 24.9455,C -1.7056,E1 25.1073,E2 497.6394} C_DIS
LIN {X 75.2931,Y -77.1641,Z 106,A -49.2351,B 24.9447,C -1.7184,E1 25.1129,E2 494.9045} C_DIS
LIN {X 77.4929,Y -74.952,Z 106,A -47.7538,B 24.9449,C -1.7149,E1 25.1157,E2 493.438} C_DIS
LIN {X 80.2299,Y -72.0146,Z 106,A -45.6458,B 24.9446,C -1.7192,E1 25.1197,E2 491.3291} C_DIS
LIN {X 82.7968,Y -69.0482,Z 106,A -43.5586,B 24.9443,C -1.7247,E1 25.1235,E2 489.2384} C_DIS
LIN {X 84.4663,Y -66.9955,Z 106,A -42.1604,B 24.944,C -1.7281,E1 25.126,E2 487.8386} C_DIS
LIN {X 86.0851,Y -64.9024,Z 106,A -40.7623,B 24.9438,C -1.7316,E1 25.1283,E2 486.439} C_DIS
LIN {X 88.1452,Y -62.0788,Z 106,A -38.7518,B 24.943,C -1.7434,E1 25.1316,E2 484.4104} C_DIS
LIN {X 90.0196,Y -59.3245,Z 106,A -37.122,B 24.9431,C -1.7422,E1 25.1341,E2 482.7914} C_DIS
LIN {X 91.786,Y -56.5569,Z 106,A -35.2537,B 24.9424,C -1.7526,E1 25.1369,E2 480.908} C_DIS
LIN {X 93.3824,Y -53.8766,Z 106,A -33.7738,B 24.9426,C -1.7496,E1 25.139,E2 479.4428} C_DIS
LIN {X 94.7089,Y -51.5089,Z 106,A -32.2696,B 24.9422,C -1.7566,E1 25.141,E2 477.93} C_DIS
LIN {X 96.3,Y -48.4734,Z 106,A -30.363,B 24.9416,C -1.7657,E1 25.1435,E2 476.012} C_DIS
LIN {X 98.0189,Y -44.896,Z 106,A -28.4351,B 24.9416,C -1.7641,E1 25.1458,E2 474.0982} C_DIS
LIN {X 99.0912,Y -42.4769,Z 106,A -27.038,B 24.9414,C -1.768,E1 25.1473,E2 472.6996} C_DIS
LIN {X 100.1038,Y -40.0323,Z 106,A -25.6411,B 24.9412,C -1.772,E1 25.1488,E2 471.3011} C_DIS
LIN {X 101.1413,Y -37.3299,Z 106,A -24.0379,B 24.9406,C -1.7796,E1 25.1504,E2 469.6888} C_DIS
LIN {X 102.3702,Y -33.8186,Z 106,A -22.0287,B 24.9401,C -1.7872,E1 25.1522,E2 467.673} C_DIS
LIN {X 103.3041,Y -30.8419,Z 106,A -20.5025,B 24.9401,C -1.7867,E1 25.1534,E2 466.1568} C_DIS
LIN {X 104.3693,Y -27.0187,Z 106,A -18.6356,B 24.9404,C -1.7827,E1 25.1548,E2 464.31} C_DIS
LIN {X 105.0009,Y -24.4492,Z 106,A -17.2387,B 24.9402,C -1.7868,E1 25.1557,E2 462.9116} C_DIS
LIN {X 105.474,Y -22.329,Z 106,A -15.7867,B 24.939,C -1.8036,E1 25.1566,E2 461.4284} C_DIS
LIN {X 106.0824,Y -19.2214,Z 106,A -14.2073,B 24.939,C -1.8045,E1 25.1574,E2 459.8561} C_DIS
LIN {X 106.6448,Y -15.8193,Z 106,A -12.2052,B 24.9381,C -1.8178,E1 25.1583,E2 457.8343} C_DIS
LIN {X 107.1548,Y -11.8832,Z 106,A -10.1105,B 24.9376,C -1.824,E1 25.159,E2 455.7373} C_DIS
LIN {X 107.5196,Y -7.9311,Z 106,A -8.1837,B 24.9377,C -1.8228,E1 25.1594,E2 453.8248} C_DIS
LIN {X 107.7022,Y -4.8168,Z 106,A -6.7656,B 24.9381,C -1.8176,E1 25.1596,E2 452.4273} C_DIS
LIN {X 107.7879,Y -2.1722,Z 106,A -5.1297,B 24.9371,C -1.8323,E1 25.1598,E2 450.7665} C_DIS
LIN {X 107.8072,Y 0.7789,Z 106,A -3.4998,B 24.9365,C -1.8401,E1 25.1598,E2 449.128} C_DIS
LIN {X 107.7386,Y 3.9682,Z 106,A -1.8994,B 24.9365,C -1.8414,E1 25.1596,E2 447.5341} C_DIS
LIN {X 107.5768,Y 7.0838,Z 106,A -0.4809,B 24.9368,C -1.8362,E1 25.1594,E2 446.1363} C_DIS
LIN {X 107.4141,Y 9.2499,Z 106,A 1.0614,B 24.9354,C -1.8569,E1 25.1591,E2 444.5542} C_DIS
LIN {X 107.1548,Y 11.8832,Z 106,A 2.4483,B 24.9351,C -1.8606,E1 25.1586,E2 443.1669} C_DIS
LIN {X 106.6448,Y 15.8193,Z 106,A 4.5529,B 24.9347,C -1.8671,E1 25.1578,E2 441.0594} C_DIS
LIN {X 106.1229,Y 18.9962,Z 106,A 6.1469,B 24.9347,C -1.8673,E1 25.1571,E2 439.4741} C_DIS
LIN {X 105.474,Y 22.329,Z 106,A 8.073,B 24.9339,C -1.8783,E1 25.156,E2 437.5334} C_DIS
LIN {X 104.5807,Y 26.1961,Z 106,A 10.1403,B 24.9335,C -1.883,E1 25.1546,E2 435.467} C_DIS
LIN {X 103.9063,Y 28.7547,Z 106,A 11.4309,B 24.9335,C -1.8822,E1 25.1537,E2 434.1856} C_DIS
LIN {X 102.7775,Y 32.5598,Z 106,A 13.4652,B 24.9334,C -1.8853,E1 25.152,E2 432.1556} C_DIS
LIN {X 101.7907,Y 35.5193,Z 106,A 15.1123,B 24.933,C -1.8898,E1 25.1506,E2 430.5071} C_DIS
LIN {X 100.4143,Y 39.2418,Z 106,A 17.2082,B 24.9326,C -1.8955,E1 25.1485,E2 428.4095} C_DIS
LIN {X 99.357,Y 41.8463,Z 106,A 18.6458,B 24.9326,C -1.8974,E1 25.147,E2 426.9754} C_DIS
LIN {X 97.819,Y 45.3255,Z 106,A 20.4738,B 24.9326,C -1.8948,E1 25.1449,E2 425.1636} C_DIS
LIN {X 96.8876,Y 47.288,Z 106,A 22.0177,B 24.9313,C -1.9149,E1 25.143,E2 423.5803} C_DIS
LIN {X 95.0814,Y 50.8221,Z 106,A 24.1144,B 24.9309,C -1.9202,E1 25.1403,E2 421.4822} C_DIS
LIN {X 93.1464,Y 54.2873,Z 106,A 26.0435,B 24.931,C -1.9181,E1 25.1376,E2 419.5682} C_DIS
LIN {X 91.535,Y 56.9587,Z 106,A 27.6916,B 24.9307,C -1.9221,E1 25.1352,E2 417.9189} C_DIS
LIN {X 90.1096,Y 59.1879,Z 106,A 29.1654,B 24.9303,C -1.9287,E1 25.133,E2 416.437} C_DIS
LIN {X 88.1452,Y 62.0788,Z 106,A 30.9378,B 24.9302,C -1.9297,E1 25.1302,E2 414.671} C_DIS
LIN {X 86.5952,Y 64.2233,Z 106,A 32.5046,B 24.9294,C -1.9401,E1 25.1275,E2 413.0871} C_DIS
LIN {X 84.993,Y 66.3292,Z 106,A 33.9036,B 24.9292,C -1.9432,E1 25.1252,E2 411.6873} C_DIS
LIN {X 83.3396,Y 68.395,Z 106,A 35.3026,B 24.929,C -1.9463,E1 25.1227,E2 410.2876} C_DIS
LIN {X 80.7657,Y 71.4162,Z 106,A 37.4015,B 24.9287,C -1.9507,E1 25.1188,E2 408.1878} C_DIS
LIN {X 78.6641,Y 73.7218,Z 106,A 38.9453,B 24.9287,C -1.9495,E1 25.1159,E2 406.6535} C_DIS
LIN {X 76.5673,Y 75.8973,Z 106,A 40.5419,B 24.9285,C -1.9526,E1 25.1128,E2 405.0564} C_DIS
LIN {X 73.3767,Y 78.9887,Z 106,A 42.8321,B 24.9284,C -1.9545,E1 25.1082,E2 402.7713} C_DIS
LIN {X 71.0941,Y 81.047,Z 106,A 44.4731,B 24.9281,C -1.9581,E1 25.1048,E2 401.1283} C_DIS
LIN {X 68.395,Y 83.3396,Z 106,A 46.333,B 24.9279,C -1.9607,E1 25.1008,E2 399.2693} C_DIS
LIN {X 66.3292,Y 84.993,Z 106,A 47.9019,B 24.9272,C -1.9702,E1 25.0973,E2 397.6838} C_DIS
LIN {X 64.2233,Y 86.5952,Z 106,A 49.303,B 24.9271,C -1.9725,E1 25.0942,E2 396.2823} C_DIS
LIN {X 60.9925,Y 88.9004,Z 106,A 51.4046,B 24.9268,C -1.9757,E1 25.0893,E2 394.1804} C_DIS
LIN {X 58.7924,Y 90.3704,Z 106,A 52.6374,B 24.9272,C -1.9707,E1 25.0865,E2 392.9635} C_DIS
LIN {X 56.1521,Y 92.0321,Z 106,A 54.2898,B 24.927,C -1.973,E1 25.0826,E2 391.3109} C_DIS
LIN {X 53.1402,Y 93.8055,Z 106,A 56.3104,B 24.9263,C -1.9825,E1 25.0777,E2 389.2739} C_DIS
LIN {X 50.3797,Y 95.3144,Z 106,A 57.8226,B 24.9266,C -1.9781,E1 25.074,E2 387.7764} C_DIS
LIN {X 47.7124,Y 96.6772,Z 106,A 59.4566,B 24.9264,C -1.9819,E1 25.0699,E2 386.1379} C_DIS
LIN {X 44.4482,Y 98.2207,Z 106,A 61.0726,B 24.9271,C -1.9716,E1 25.0659,E2 384.5504} C_DIS
LIN {X 42.4769,Y 99.0912,Z 106,A 62.6217,B 24.9258,C -1.9896,E1 25.0618,E2 382.9624} C_DIS
LIN {X 38.8009,Y 100.5875,Z 106,A 64.5578,B 24.9262,C -1.9845,E1 25.0568,E2 381.0427} C_DIS
LIN {X 35.8736,Y 101.6663,Z 106,A 66.2123,B 24.9261,C -1.986,E1 25.0525,E2 379.3883} C_DIS
LIN {X 32.1073,Y 102.9178,Z 106,A 68.3885,B 24.9257,C -1.9904,E1 25.0467,E2 377.2056} C_DIS
LIN {X 28.7548,Y 103.9063,Z 106,A 70.3418,B 24.9253,C -1.9956,E1 25.0414,E2 375.2432} C_DIS
LIN {X 25.7359,Y 104.693,Z 106,A 71.8285,B 24.9258,C -1.9896,E1 25.0374,E2 373.7729} C_DIS
LIN {X 21.8649,Y 105.5692,Z 106,A 73.7006,B 24.9264,C -1.981,E1 25.0324,E2 371.9238} C_DIS
LIN {X 19.2676,Y 106.0741,Z 106,A 75.3405,B 24.9257,C -1.9911,E1 25.0278,E2 370.2618} C_DIS
LIN {X 15.8193,Y 106.6448,Z 106,A 77.3663,B 24.9251,C -1.9985,E1 25.0222,E2 368.2206} C_DIS
LIN {X 11.8832,Y 107.1548,Z 106,A 79.4748,B 24.9251,C -1.9988,E1 25.0163,E2 366.1127} C_DIS
LIN {X 7.9311,Y 107.5196,Z 106,A 81.4146,B 24.9256,C -1.9921,E1 25.011,E2 364.1899} C_DIS
LIN {X 4.8168,Y 107.7022,Z 106,A 83.0554,B 24.9256,C -1.9914,E1 25.0064,E2 362.5513} C_DIS
LIN {X 1.323,Y 107.8036,Z 106,A 85.1001,B 24.9251,C -1.9987,E1 25.0007,E2 360.4897} C_DIS
LIN {X -1.323,Y 107.8036,Z 106,A 86.5071,B 24.9251,C -1.9984,E1 24.9968,E2 359.0834} C_DIS
LIN {X -3.9682,Y 107.7386,Z 106,A 87.9144,B 24.9251,C -1.998,E1 24.9928,E2 357.6769} C_DIS
LIN {X -7.0838,Y 107.5768,Z 106,A 89.3721,B 24.9258,C -1.9894,E1 24.9888,E2 356.2391} C_DIS
LIN {X -11.8832,Y 107.1548,Z 106,A 91.9678,B 24.9258,C -1.9894,E1 24.9816,E2 353.6418} C_DIS
LIN {X -14.9784,Y 106.7642,Z 106,A 93.3977,B 24.9265,C -1.9795,E1 24.9777,E2 352.2346} C_DIS
LIN {X -17.1268,Y 106.4426,Z 106,A 94.9718,B 24.9254,C -1.9952,E1 24.9732,E2 350.6217} C_DIS
LIN {X -20.199,Y 105.9007,Z 106,A 96.445,B 24.926,C -1.9867,E1 24.9693,E2 349.1673} C_DIS
LIN {X -23.6217,Y 105.1921,Z 106,A 98.4756,B 24.9256,C -1.9918,E1 24.9637,E2 347.1219} C_DIS
LIN {X -26.5288,Y 104.4952,Z 106,A 99.9409,B 24.9261,C -1.9855,E1 24.9597,E2 345.6697} C_DIS
LIN {X -30.0277,Y 103.5456,Z 106,A 101.9992,B 24.9259,C -1.9886,E1 24.9542,E2 343.6008} C_DIS
LIN {X -33.3023,Y 102.5373,Z 106,A 103.7317,B 24.9263,C -1.983,E1 24.9496,E2 341.8784} C_DIS
LIN {X -36.7657,Y 101.3471,Z 106,A 105.6067,B 24.9267,C -1.9778,E1 24.9447,E2 340.0122} C_DIS
LIN {X -39.2418,Y 100.4143,Z 106,A 107.0171,B 24.9267,C -1.9761,E1 24.941,E2 338.6029} C_DIS
LIN {X -41.6943,Y 99.421,Z 106,A 108.4275,B 24.9269,C -1.9742,E1 24.9374,E2 337.1937} C_DIS
LIN {X -44.896,Y 98.0189,Z 106,A 110.2912,B 24.9271,C -1.9717,E1 24.9326,E2 335.3315} C_DIS
LIN {X -47.7124,Y 96.6772,Z 106,A 111.9549,B 24.9273,C -1.9693,E1 24.9284,E2 333.6692} C_DIS
LIN {X -50.8221,Y 95.0814,Z 106,A 113.8193,B 24.9275,C -1.9664,E1 24.9238,E2 331.8065} C_DIS
LIN {X -53.1402,Y 93.8055,Z 106,A 115.2309,B 24.9277,C -1.9642,E1 24.9204,E2 330.3961} C_DIS
LIN {X -55.4263,Y 92.4732,Z 106,A 116.6429,B 24.9278,C -1.9619,E1 24.917,E2 328.9854} C_DIS
LIN {X -58.0777,Y 90.8292,Z 106,A 118.1413,B 24.9285,C -1.9527,E1 24.9135,E2 327.5041} C_DIS
LIN {X -60.2892,Y 89.3765,Z 106,A 119.6867,B 24.9283,C -1.9552,E1 24.9099,E2 325.9476} C_DIS
LIN {X -63.1559,Y 87.3768,Z 106,A 121.5857,B 24.9285,C -1.953,E1 24.9055,E2 324.0473} C_DIS
LIN {X -65.2812,Y 85.8005,Z 106,A 122.9983,B 24.9287,C -1.9503,E1 24.9024,E2 322.6361} C_DIS
LIN {X -67.4351,Y 84.1176,Z 106,A 124.415,B 24.929,C -1.9458,E1 24.8993,E2 321.2248} C_DIS
LIN {X -69.7732,Y 82.1867,Z 106,A 125.846,B 24.9298,C -1.9354,E1 24.8963,E2 319.8131} C_DIS
LIN {X -71.7789,Y 80.4409,Z 106,A 127.4932,B 24.9294,C -1.941,E1 24.8928,E2 318.146} C_DIS
LIN {X -74.3405,Y 78.0823,Z 106,A 129.5277,B 24.9292,C -1.9436,E1 24.8886,E2 316.0971} C_DIS
LIN {X -76.5673,Y 75.8973,Z 106,A 131.0241,B 24.9299,C -1.9335,E1 24.8857,E2 314.6183} C_DIS
LIN {X -78.9887,Y 73.3767,Z 106,A 133.062,B 24.9298,C -1.9357,E1 24.8817,E2 312.5664} C_DIS
LIN {X -81.636,Y 70.4197,Z 106,A 135.1833,B 24.9301,C -1.9307,E1 24.8778,E2 310.4474} C_DIS
LIN {X -83.6378,Y 68.027,Z 106,A 136.6804,B 24.9309,C -1.9204,E1 24.8752,E2 308.9681} C_DIS
LIN {X -86.0851,Y 64.9024,Z 106,A 138.8022,B 24.9312,C -1.9152,E1 24.8716,E2 306.8485} C_DIS
LIN {X -88.1452,Y 62.0788,Z 106,A 140.6709,B 24.9316,C -1.9105,E1 24.8685,E2 304.9819} C_DIS
LIN {X -89.6421,Y 59.897,Z 106,A 142.0855,B 24.9318,C -1.9069,E1 24.8663,E2 303.5689} C_DIS
LIN {X -91.0851,Y 57.679,Z 106,A 143.5007,B 24.9321,C -1.9033,E1 24.8642,E2 302.1552} C_DIS
LIN {X -92.4732,Y 55.4263,Z 106,A 144.9156,B 24.9324,C -1.8995,E1 24.8621,E2 300.7418} C_DIS
LIN {X -93.8055,Y 53.1402,Z 106,A 146.4591,B 24.9323,C -1.9006,E1 24.86,E2 299.1878} C_DIS
LIN {X -95.0814,Y 50.8221,Z 106,A 147.9163,B 24.9324,C -1.8984,E1 24.8581,E2 297.7283} C_DIS
LIN {X -96.3,Y 48.4734,Z 106,A 149.3315,B 24.9327,C -1.8945,E1 24.8563,E2 296.3146} C_DIS
LIN {X -98.0189,Y 44.896,Z 106,A 151.3229,B 24.9335,C -1.8838,E1 24.8539,E2 294.338} C_DIS
LIN {X -99.2752,Y 42.0404,Z 106,A 152.8771,B 24.9341,C -1.8749,E1 24.8522,E2 292.7964} C_DIS
LIN {X -100.1038,Y 40.0323,Z 106,A 154.2862,B 24.9337,C -1.8808,E1 24.8507,E2 291.3654} C_DIS
LIN {X -101.2184,Y 37.1185,Z 106,A 155.785,B 24.9345,C -1.8698,E1 24.8493,E2 289.8844} C_DIS
LIN {X -102.3702,Y 33.8186,Z 106,A 157.8257,B 24.9344,C -1.8707,E1 24.8474,E2 287.8298} C_DIS
LIN {X -103.3041,Y 30.8419,Z 106,A 159.4018,B 24.935,C -1.8625,E1 24.8462,E2 286.2642} C_DIS
LIN {X -104.2514,Y 27.4775,Z 106,A 161.1949,B 24.9356,C -1.8542,E1 24.8448,E2 284.4805} C_DIS
LIN {X -105.0009,Y 24.4492,Z 106,A 162.8645,B 24.9359,C -1.8494,E1 24.8437,E2 282.8126} C_DIS
LIN {X -105.7644,Y 20.907,Z 106,A 164.9246,B 24.9359,C -1.8481,E1 24.8426,E2 280.7432} C_DIS
LIN {X -106.2244,Y 18.4317,Z 106,A 166.3217,B 24.9361,C -1.846,E1 24.8419,E2 279.343} C_DIS
LIN {X -106.6448,Y 15.8193,Z 106,A 167.7378,B 24.9364,C -1.8418,E1 24.8413,E2 277.9283} C_DIS
LIN {X -107.0851,Y 12.4785,Z 106,A 169.4351,B 24.937,C -1.8326,E1 24.8407,E2 276.243} C_DIS
LIN {X -107.4141,Y 9.2499,Z 106,A 171.1077,B 24.9376,C -1.8251,E1 24.8403,E2 274.5783} C_DIS
LIN {X -107.6088,Y 6.6111,Z 106,A 172.6945,B 24.9374,C -1.8272,E1 24.84,E2 272.9768} C_DIS
LIN {X -107.7386,Y 3.9682,Z 106,A 174.1106,B 24.9377,C -1.823,E1 24.8399,E2 271.5622} C_DIS
LIN {X -107.808,Y 0.6273,Z 106,A 175.8316,B 24.9382,C -1.8153,E1 24.8398,E2 269.8493} C_DIS
LIN {X -107.7647,Y -3.1194,Z 106,A 177.5024,B 24.9395,C -1.797,E1 24.8398,E2 268.2122} C_DIS
LIN {X -107.6557,Y -5.7631,Z 106,A 179.15,B 24.9392,C -1.8014,E1 24.8401,E2 266.5441} C_DIS
LIN {X -107.4141,Y -9.25,Z 106,A -178.8088,B 24.9392,C -1.8022,E1 24.8405,E2 264.4886} C_DIS
LIN {X -107.1548,Y -11.8832,Z 106,A -177.5632,B 24.9398,C -1.7918,E1 24.8409,E2 263.2605} C_DIS
LIN {X -106.7642,Y -14.9784,Z 106,A -176.1252,B 24.9407,C -1.7784,E1 24.8414,E2 261.8459} C_DIS
LIN {X -106.4426,Y -17.1268,Z 106,A -174.5609,B 24.94,C -1.7899,E1 24.8421,E2 260.2447} C_DIS
LIN {X -105.9007,Y -20.199,Z 106,A -173.0619,B 24.9407,C -1.7788,E1 24.8428,E2 258.7633} C_DIS
LIN {X -105.1921,Y -23.6217,Z 106,A -171.0215,B 24.9407,C -1.7798,E1 24.844,E2 256.7085} C_DIS
LIN {X -104.5807,Y -26.1961,Z 106,A -169.6056,B 24.9409,C -1.7759,E1 24.845,E2 255.2937} C_DIS
LIN {X -103.9063,Y -28.7548,Z 106,A -168.2402,B 24.9413,C -1.77,E1 24.846,E2 253.9344} C_DIS
LIN {X -103.029,Y -31.7486,Z 106,A -166.6914,B 24.9419,C -1.7609,E1 24.8472,E2 252.3983} C_DIS
LIN {X -101.9475,Y -35.0723,Z 106,A -164.6513,B 24.9419,C -1.7622,E1 24.8491,E2 250.3436} C_DIS
LIN {X -100.8883,Y -38.0066,Z 106,A -163.0966,B 24.9424,C -1.7534,E1 24.8505,E2 248.801} C_DIS
LIN {X -99.9252,Y -40.4711,Z 106,A -161.7378,B 24.9428,C -1.7475,E1 24.8519,E2 247.4486} C_DIS
LIN {X -98.9019,Y -42.9112,Z 106,A -160.3226,B 24.943,C -1.7438,E1 24.8535,E2 246.0345} C_DIS
LIN {X -97.4606,Y -46.0954,Z 106,A -158.2832,B 24.943,C -1.7454,E1 24.8559,E2 243.9802} C_DIS
LIN {X -96.0195,Y -49.0222,Z 106,A -156.7509,B 24.9437,C -1.733,E1 24.8578,E2 242.4692} C_DIS
LIN {X -94.4506,Y -51.985,Z 106,A -154.9166,B 24.9439,C -1.73,E1 24.8602,E2 240.6323} C_DIS
LIN {X -92.863,Y -54.7667,Z 106,A -153.137,B 24.944,C -1.7284,E1 24.8627,E2 238.8472} C_DIS
LIN {X -91.0851,Y -57.679,Z 106,A -151.3808,B 24.9445,C -1.7214,E1 24.8653,E2 237.0987} C_DIS
LIN {X -89.3765,Y -60.2892,Z 106,A -149.7137,B 24.9447,C -1.7176,E1 24.8679,E2 235.4325} C_DIS
LIN {X -87.3768,Y -63.1559,Z 106,A -147.8457,B 24.945,C -1.7133,E1 24.8709,E2 233.5656} C_DIS
LIN {X -85.8005,Y -65.2812,Z 106,A -146.432,B 24.9452,C -1.7101,E1 24.8733,E2 232.1526} C_DIS
LIN {X -83.8313,Y -67.7883,Z 106,A -144.6572,B 24.9452,C -1.7092,E1 24.8764,E2 230.3717} C_DIS
LIN {X -81.636,Y -70.4197,Z 106,A -142.7283,B 24.9452,C -1.709,E1 24.8799,E2 228.4343} C_DIS
LIN {X -79.5629,Y -72.751,Z 106,A -141.3806,B 24.9463,C -1.6934,E1 24.8823,E2 227.1177} C_DIS
LIN {X -77.1641,Y -75.2931,Z 106,A -139.196,B 24.9457,C -1.7019,E1 24.8866,E2 224.9035} C_DIS
LIN {X -74.952,Y -77.4929,Z 106,A -137.7001,B 24.9463,C -1.6922,E1 24.8895,E2 223.4245} C_DIS
LIN {X -72.3816,Y -79.9014,Z 106,A -135.6559,B 24.9462,C -1.6951,E1 24.8938,E2 221.3653} C_DIS
LIN {X -70.4197,Y -81.636,Z 106,A -134.2524,B 24.9462,C -1.6928,E1 24.8967,E2 219.9616} C_DIS
LIN {X -68.027,Y -83.6378,Z 106,A -132.7574,B 24.9469,C -1.6834,E1 24.8999,E2 218.4833} C_DIS
LIN {X -65.9539,Y -85.2821,Z 106,A -131.3457,B 24.947,C -1.681,E1 24.903,E2 217.072} C_DIS
LIN {X -63.1559,Y -87.3768,Z 106,A -129.4811,B 24.9472,C -1.6781,E1 24.9072,E2 215.2078} C_DIS
LIN {X -60.9925,Y -88.9004,Z 106,A -127.9001,B 24.9469,C -1.6826,E1 24.9109,E2 213.6108} C_DIS
LIN {X -58.509,Y -90.5523,Z 106,A -126.4135,B 24.9473,C -1.6762,E1 24.9143,E2 212.1344} C_DIS
LIN {X -56.1521,Y -92.0321,Z 106,A -124.9953,B 24.9476,C -1.6716,E1 24.9177,E2 210.7228} C_DIS
Enddeposition()
END
